gfCNCPoint1[8476] = {X 60.5656, Y 8.0531, Z -1.3333, A 0.000, B 0.000, C 0.000 }
gfCNCPoint1[8477] = {X 61.4618, Y 8.3667, Z -1.3333, A 0.000, B 0.000, C 0.000 }
gfCNCPoint1[8478] = {X 62.2657, Y 8.8718, Z -1.3333, A 0.000, B 0.000, C 0.000 }
gfCNCPoint1[8479] = {X 62.9371, Y 9.5432, Z -1.3333, A 0.000, B 0.000, C 0.000 }
gfCNCPoint1[8480] = {X 63.4422, Y 10.3471, Z -1.3333, A 0.000, B 0.000, C 0.000 }
gfCNCPoint1[8481] = {X 63.7558, Y 11.2433, Z -1.3333, A 0.000, B 0.000, C 0.000 }
gfCNCPoint1[8482] = {X 63.8621, Y 12.1868, Z -1.3333, A 0.000, B 0.000, C 0.000 }
gfCNCPoint1[8483] = {X 63.8621, Y 12.9781, Z -1.3333, A 0.000, B 0.000, C 0.000 }
gfCNCPoint1[8484] = {X 63.7771, Y 13.8227, Z -1.3333, A 0.000, B 0.000, C 0.000 }
gfCNCPoint1[8485] = {X 63.5256, Y 14.6335, Z -1.3333, A 0.000, B 0.000, C 0.000 }
gfCNCPoint1[8486] = {X 63.1176, Y 15.3779, Z -1.3333, A 0.000, B 0.000, C 0.000 }
gfCNCPoint1[8487] = {X 63.3949, Y 16.1022, Z -1.3333, A 0.000, B 0.000, C 0.000 }
gfCNCPoint1[8488] = {X 65.9589, Y 22.9155, Z -1.3333, A 0.000, B 0.000, C 0.000 }
gfCNCPoint1[8489] = {X 72.1337, Y 39.5291, Z -1.3333, A 0.000, B 0.000, C 0.000 }
gfCNCPoint1[8490] = {X 72.4511, Y 40.3274, Z -1.3333, A 0.000, B 0.000, C 0.000 }
gfCNCPoint1[8491] = {X 73.2892, Y 40.8174, Z -1.3333, A 0.000, B 0.000, C 0.000 }
gfCNCPoint1[8492] = {X 73.9939, Y 41.4851, Z -1.3333, A 0.000, B 0.000, C 0.000 }
gfCNCPoint1[8493] = {X 74.5283, Y 42.2956, Z -1.3333, A 0.000, B 0.000, C 0.000 }
gfCNCPoint1[8494] = {X 74.8643, Y 43.2065, Z -1.3333, A 0.000, B 0.000, C 0.000 }
gfCNCPoint1[8495] = {X 74.9843, Y 44.1699, Z -1.3333, A 0.000, B 0.000, C 0.000 }
gfCNCPoint1[8496] = {X 74.9845, Y 45.0000, Z -1.3333, A 0.000, B 0.000, C 0.000 }
gfCNCPoint1[8497] = {X 74.8782, Y 45.9435, Z -1.3333, A 0.000, B 0.000, C 0.000 }
gfCNCPoint1[8498] = {X 74.5646, Y 46.8397, Z -1.3333, A 0.000, B 0.000, C 0.000 }
gfCNCPoint1[8499] = {X 74.0594, Y 47.6436, Z -1.3333, A 0.000, B 0.000, C 0.000 }
gfCNCPoint1[8500] = {X 73.3881, Y 48.3150, Z -1.3333, A 0.000, B 0.000, C 0.000 }
gfCNCPoint1[8501] = {X 72.5841, Y 48.8201, Z -1.3333, A 0.000, B 0.000, C 0.000 }
gfCNCPoint1[8502] = {X 71.6879, Y 49.1337, Z -1.3333, A 0.000, B 0.000, C 0.000 }
gfCNCPoint1[8503] = {X 70.7445, Y 49.2400, Z -1.3333, A 0.000, B 0.000, C 0.000 }
gfCNCPoint1[8504] = {X 64.1851, Y 49.2400, Z -1.3333, A 0.000, B 0.000, C 0.000 }
gfCNCPoint1[8505] = {X 63.2416, Y 49.1337, Z -1.3333, A 0.000, B 0.000, C 0.000 }
gfCNCPoint1[8506] = {X 62.3455, Y 48.8201, Z -1.3333, A 0.000, B 0.000, C 0.000 }
gfCNCPoint1[8507] = {X 61.5415, Y 48.3150, Z -1.3333, A 0.000, B 0.000, C 0.000 }
gfCNCPoint1[8508] = {X 60.8702, Y 47.6436, Z -1.3333, A 0.000, B 0.000, C 0.000 }
gfCNCPoint1[8509] = {X 60.3650, Y 46.8397, Z -1.3333, A 0.000, B 0.000, C 0.000 }
gfCNCPoint1[8510] = {X 60.0514, Y 45.9435, Z -1.3333, A 0.000, B 0.000, C 0.000 }
gfCNCPoint1[8511] = {X 59.9451, Y 45.0000, Z -1.3333, A 0.000, B 0.000, C 0.000 }
gfCNCPoint1[8512] = {X 59.9451, Y 44.2085, Z -1.3333, A 0.000, B 0.000, C 0.000 }
gfCNCPoint1[8513] = {X 60.0333, Y 43.3524, Z -1.3333, A 0.000, B 0.000, C 0.000 }
gfCNCPoint1[8514] = {X 60.2925, Y 42.5318, Z -1.3333, A 0.000, B 0.000, C 0.000 }
gfCNCPoint1[8515] = {X 60.7121, Y 41.7805, Z -1.3333, A 0.000, B 0.000, C 0.000 }
gfCNCPoint1[8516] = {X 60.0634, Y 40.0092, Z -1.3333, A 0.000, B 0.000, C 0.000 }
gfCNCPoint1[8517] = {X 52.0206, Y 40.0092, Z -1.3333, A 0.000, B 0.000, C 0.000 }
gfCNCPoint1[8518] = {X 51.2452, Y 42.0920, Z -1.3333, A 0.000, B 0.000, C 0.000 }
gfCNCPoint1[8519] = {X 51.2680, Y 42.1293, Z -1.3333, A 0.000, B 0.000, C 0.000 }
gfCNCPoint1[8520] = {X 51.5637, Y 42.7765, Z -1.3333, A 0.000, B 0.000, C 0.000 }
gfCNCPoint1[8521] = {X 51.7470, Y 43.4641, Z -1.3333, A 0.000, B 0.000, C 0.000 }
gfCNCPoint1[8522] = {X 51.8128, Y 44.1726, Z -1.3333, A 0.000, B 0.000, C 0.000 }
gfCNCPoint1[8523] = {X 51.8129, Y 45.0000, Z -1.3333, A 0.000, B 0.000, C 0.000 }
gfCNCPoint1[8524] = {X 51.7066, Y 45.9435, Z -1.3333, A 0.000, B 0.000, C 0.000 }
gfCNCPoint1[8525] = {X 51.3930, Y 46.8397, Z -1.3333, A 0.000, B 0.000, C 0.000 }
gfCNCPoint1[8526] = {X 50.8879, Y 47.6436, Z -1.3333, A 0.000, B 0.000, C 0.000 }
gfCNCPoint1[8527] = {X 50.2165, Y 48.3150, Z -1.3333, A 0.000, B 0.000, C 0.000 }
gfCNCPoint1[8528] = {X 49.4126, Y 48.8201, Z -1.3333, A 0.000, B 0.000, C 0.000 }
gfCNCPoint1[8529] = {X 48.5164, Y 49.1337, Z -1.3333, A 0.000, B 0.000, C 0.000 }
gfCNCPoint1[8530] = {X 47.5729, Y 49.2400, Z -1.3333, A 0.000, B 0.000, C 0.000 }
gfCNCPoint1[8531] = {X 40.6393, Y 49.2400, Z -1.3333, A 0.000, B 0.000, C 0.000 }
gfCNCPoint1[8532] = {X 39.6958, Y 49.1337, Z -1.3333, A 0.000, B 0.000, C 0.000 }
gfCNCPoint1[8533] = {X 38.7996, Y 48.8201, Z -1.3333, A 0.000, B 0.000, C 0.000 }
gfCNCPoint1[8534] = {X 37.9957, Y 48.3150, Z -1.3333, A 0.000, B 0.000, C 0.000 }
gfCNCPoint1[8535] = {X 37.3243, Y 47.6436, Z -1.3333, A 0.000, B 0.000, C 0.000 }
gfCNCPoint1[8536] = {X 36.8192, Y 46.8397, Z -1.3333, A 0.000, B 0.000, C 0.000 }
gfCNCPoint1[8537] = {X 36.5056, Y 45.9435, Z -1.3333, A 0.000, B 0.000, C 0.000 }
gfCNCPoint1[8538] = {X 36.3993, Y 45.0000, Z -1.3333, A 0.000, B 0.000, C 0.000 }
gfCNCPoint1[8539] = {X 36.3993, Y 44.2086, Z -1.3333, A 0.000, B 0.000, C 0.000 }
gfCNCPoint1[8540] = {X 36.5154, Y 43.2237, Z -1.3333, A 0.000, B 0.000, C 0.000 }
gfCNCPoint1[8541] = {X 36.8572, Y 42.2926, Z -1.3333, A 0.000, B 0.000, C 0.000 }
gfCNCPoint1[8542] = {X 37.4059, Y 41.4664, Z -1.3333, A 0.000, B 0.000, C 0.000 }
gfCNCPoint1[8543] = {X 38.1315, Y 40.7903, Z -1.3333, A 0.000, B 0.000, C 0.000 }
gfCNCPoint1[8544] = {X 38.9944, Y 40.3012, Z -1.3333, A 0.000, B 0.000, C 0.000 }
gfCNCPoint1[8545] = {X 39.5929, Y 38.8890, Z -1.3333, A 0.000, B 0.000, C 0.000 }
gfCNCPoint1[8546] = {X 40.1409, Y 37.4565, Z -1.3333, A 0.000, B 0.000, C 0.000 }
gfCNCPoint1[8547] = {X 43.7241, Y 27.8349, Z -1.3333, A 0.000, B 0.000, C 0.000 }
gfCNCPoint1[8548] = {X 39.9756, Y 26.4389, Z -1.3333, A 0.000, B 0.000, C 0.000 }
gfCNCPoint1[8549] = {X 43.7991, Y 27.8628, Z -1.3333, A 0.000, B 0.000, C 0.000 }
gfCNCPoint1[8550] = {X 48.4687, Y 15.3238, Z -1.3333, A 0.000, B 0.000, C 0.000 }
gfCNCPoint1[8551] = {X 48.0765, Y 14.6072, Z -1.3333, A 0.000, B 0.000, C 0.000 }
gfCNCPoint1[8552] = {X 47.8320, Y 13.8278, Z -1.3333, A 0.000, B 0.000, C 0.000 }
gfCNCPoint1[8553] = {X 47.7444, Y 13.0157, Z -1.3333, A 0.000, B 0.000, C 0.000 }
gfCNCPoint1[8554] = {X 47.7442, Y 12.1868, Z -1.3333, A 0.000, B 0.000, C 0.000 }
gfCNCPoint1[8555] = {X 47.8485, Y 11.2611, Z -1.3333, A 0.000, B 0.000, C 0.000 }
gfCNCPoint1[8556] = {X 48.1562, Y 10.3819, Z -1.3333, A 0.000, B 0.000, C 0.000 }
gfCNCPoint1[8557] = {X 48.6518, Y 9.5931, Z -1.3333, A 0.000, B 0.000, C 0.000 }
gfCNCPoint1[8558] = {X 49.3105, Y 8.9344, Z -1.3333, A 0.000, B 0.000, C 0.000 }
gfCNCPoint1[8559] = {X 50.0993, Y 8.4388, Z -1.3333, A 0.000, B 0.000, C 0.000 }
gfCNCPoint1[8560] = {X 50.9785, Y 8.1311, Z -1.3333, A 0.000, B 0.000, C 0.000 }
gfCNCPoint1[8561] = {X 51.9042, Y 8.0268, Z -1.3333, A 0.000, B 0.000, C 0.000 }
gfCNCPoint1[8562] = {X 59.6221, Y 8.0268, Z -1.3333, A 0.000, B 0.000, C 0.000 }
gfCNCPoint1[8563] = {X 60.5478, Y 8.1311, Z -1.3333, A 0.000, B 0.000, C 0.000 }
gfCNCPoint1[8564] = {X 61.4271, Y 8.4388, Z -1.3333, A 0.000, B 0.000, C 0.000 }
gfCNCPoint1[8565] = {X 62.2158, Y 8.9344, Z -1.3333, A 0.000, B 0.000, C 0.000 }
gfCNCPoint1[8566] = {X 62.8745, Y 9.5931, Z -1.3333, A 0.000, B 0.000, C 0.000 }
gfCNCPoint1[8567] = {X 63.3702, Y 10.3819, Z -1.3333, A 0.000, B 0.000, C 0.000 }
gfCNCPoint1[8568] = {X 63.6778, Y 11.2611, Z -1.3333, A 0.000, B 0.000, C 0.000 }
gfCNCPoint1[8569] = {X 63.7821, Y 12.1868, Z -1.3333, A 0.000, B 0.000, C 0.000 }
gfCNCPoint1[8570] = {X 63.7821, Y 12.9781, Z -1.3333, A 0.000, B 0.000, C 0.000 }
gfCNCPoint1[8571] = {X 63.6959, Y 13.8205, Z -1.3333, A 0.000, B 0.000, C 0.000 }
gfCNCPoint1[8572] = {X 63.4410, Y 14.6279, Z -1.3333, A 0.000, B 0.000, C 0.000 }
gfCNCPoint1[8573] = {X 63.0278, Y 15.3670, Z -1.3333, A 0.000, B 0.000, C 0.000 }
gfCNCPoint1[8574] = {X 63.3201, Y 16.1306, Z -1.3333, A 0.000, B 0.000, C 0.000 }
gfCNCPoint1[8575] = {X 65.8840, Y 22.9436, Z -1.3333, A 0.000, B 0.000, C 0.000 }
gfCNCPoint1[8576] = {X 72.0590, Y 39.5578, Z -1.3333, A 0.000, B 0.000, C 0.000 }
gfCNCPoint1[8577] = {X 72.3889, Y 40.3876, Z -1.3333, A 0.000, B 0.000, C 0.000 }
gfCNCPoint1[8578] = {X 73.2202, Y 40.8657, Z -1.3333, A 0.000, B 0.000, C 0.000 }
gfCNCPoint1[8579] = {X 73.9200, Y 41.5215, Z -1.3333, A 0.000, B 0.000, C 0.000 }
gfCNCPoint1[8580] = {X 74.4510, Y 42.3201, Z -1.3333, A 0.000, B 0.000, C 0.000 }
gfCNCPoint1[8581] = {X 74.7850, Y 43.2191, Z -1.3333, A 0.000, B 0.000, C 0.000 }
gfCNCPoint1[8582] = {X 74.9043, Y 44.1706, Z -1.3333, A 0.000, B 0.000, C 0.000 }
gfCNCPoint1[8583] = {X 74.9045, Y 45.0000, Z -1.3333, A 0.000, B 0.000, C 0.000 }
gfCNCPoint1[8584] = {X 74.8002, Y 45.9257, Z -1.3333, A 0.000, B 0.000, C 0.000 }
gfCNCPoint1[8585] = {X 74.4925, Y 46.8050, Z -1.3333, A 0.000, B 0.000, C 0.000 }
gfCNCPoint1[8586] = {X 73.9969, Y 47.5937, Z -1.3333, A 0.000, B 0.000, C 0.000 }
gfCNCPoint1[8587] = {X 73.3382, Y 48.2524, Z -1.3333, A 0.000, B 0.000, C 0.000 }
gfCNCPoint1[8588] = {X 72.5494, Y 48.7480, Z -1.3333, A 0.000, B 0.000, C 0.000 }
gfCNCPoint1[8589] = {X 71.6701, Y 49.0557, Z -1.3333, A 0.000, B 0.000, C 0.000 }
gfCNCPoint1[8590] = {X 70.7445, Y 49.1600, Z -1.3333, A 0.000, B 0.000, C 0.000 }
gfCNCPoint1[8591] = {X 64.1851, Y 49.1600, Z -1.3333, A 0.000, B 0.000, C 0.000 }
gfCNCPoint1[8592] = {X 63.2594, Y 49.0557, Z -1.3333, A 0.000, B 0.000, C 0.000 }
gfCNCPoint1[8593] = {X 62.3802, Y 48.7480, Z -1.3333, A 0.000, B 0.000, C 0.000 }
gfCNCPoint1[8594] = {X 61.5914, Y 48.2524, Z -1.3333, A 0.000, B 0.000, C 0.000 }
gfCNCPoint1[8595] = {X 60.9327, Y 47.5937, Z -1.3333, A 0.000, B 0.000, C 0.000 }
gfCNCPoint1[8596] = {X 60.4371, Y 46.8050, Z -1.3333, A 0.000, B 0.000, C 0.000 }
gfCNCPoint1[8597] = {X 60.1294, Y 45.9257, Z -1.3333, A 0.000, B 0.000, C 0.000 }
gfCNCPoint1[8598] = {X 60.0251, Y 45.0000, Z -1.3333, A 0.000, B 0.000, C 0.000 }
gfCNCPoint1[8599] = {X 60.0251, Y 44.2086, Z -1.3333, A 0.000, B 0.000, C 0.000 }
gfCNCPoint1[8600] = {X 60.1145, Y 43.3551, Z -1.3333, A 0.000, B 0.000, C 0.000 }
gfCNCPoint1[8601] = {X 60.3770, Y 42.5381, Z -1.3333, A 0.000, B 0.000, C 0.000 }
gfCNCPoint1[8602] = {X 60.8017, Y 41.7924, Z -1.3333, A 0.000, B 0.000, C 0.000 }
gfCNCPoint1[8603] = {X 60.1193, Y 39.9292, Z -1.3333, A 0.000, B 0.000, C 0.000 }
gfCNCPoint1[8604] = {X 51.9650, Y 39.9292, Z -1.3333, A 0.000, B 0.000, C 0.000 }
gfCNCPoint1[8605] = {X 51.1567, Y 42.1005, Z -1.3333, A 0.000, B 0.000, C 0.000 }
gfCNCPoint1[8606] = {X 51.1989, Y 42.1698, Z -1.3333, A 0.000, B 0.000, C 0.000 }
gfCNCPoint1[8607] = {X 51.4887, Y 42.8044, Z -1.3333, A 0.000, B 0.000, C 0.000 }
gfCNCPoint1[8608] = {X 51.6683, Y 43.4786, Z -1.3333, A 0.000, B 0.000, C 0.000 }
gfCNCPoint1[8609] = {X 51.7328, Y 44.1733, Z -1.3333, A 0.000, B 0.000, C 0.000 }
gfCNCPoint1[8610] = {X 51.7329, Y 45.0000, Z -1.3333, A 0.000, B 0.000, C 0.000 }
gfCNCPoint1[8611] = {X 51.6286, Y 45.9257, Z -1.3333, A 0.000, B 0.000, C 0.000 }
gfCNCPoint1[8612] = {X 51.3210, Y 46.8050, Z -1.3333, A 0.000, B 0.000, C 0.000 }
gfCNCPoint1[8613] = {X 50.8253, Y 47.5937, Z -1.3333, A 0.000, B 0.000, C 0.000 }
gfCNCPoint1[8614] = {X 50.1666, Y 48.2524, Z -1.3333, A 0.000, B 0.000, C 0.000 }
gfCNCPoint1[8615] = {X 49.3779, Y 48.7480, Z -1.3333, A 0.000, B 0.000, C 0.000 }
gfCNCPoint1[8616] = {X 48.4986, Y 49.0557, Z -1.3333, A 0.000, B 0.000, C 0.000 }
gfCNCPoint1[8617] = {X 47.5729, Y 49.1600, Z -1.3333, A 0.000, B 0.000, C 0.000 }
gfCNCPoint1[8618] = {X 40.6393, Y 49.1600, Z -1.3333, A 0.000, B 0.000, C 0.000 }
gfCNCPoint1[8619] = {X 39.7136, Y 49.0557, Z -1.3333, A 0.000, B 0.000, C 0.000 }
gfCNCPoint1[8620] = {X 38.8343, Y 48.7480, Z -1.3333, A 0.000, B 0.000, C 0.000 }
gfCNCPoint1[8621] = {X 38.0456, Y 48.2524, Z -1.3333, A 0.000, B 0.000, C 0.000 }
gfCNCPoint1[8622] = {X 37.3869, Y 47.5937, Z -1.3333, A 0.000, B 0.000, C 0.000 }
gfCNCPoint1[8623] = {X 36.8913, Y 46.8050, Z -1.3333, A 0.000, B 0.000, C 0.000 }
gfCNCPoint1[8624] = {X 36.5836, Y 45.9257, Z -1.3333, A 0.000, B 0.000, C 0.000 }
gfCNCPoint1[8625] = {X 36.4793, Y 45.0000, Z -1.3333, A 0.000, B 0.000, C 0.000 }
gfCNCPoint1[8626] = {X 36.4793, Y 44.2087, Z -1.3333, A 0.000, B 0.000, C 0.000 }
gfCNCPoint1[8627] = {X 36.5947, Y 43.2361, Z -1.3333, A 0.000, B 0.000, C 0.000 }
gfCNCPoint1[8628] = {X 36.9343, Y 42.3175, Z -1.3333, A 0.000, B 0.000, C 0.000 }
gfCNCPoint1[8629] = {X 37.4792, Y 41.5038, Z -1.3333, A 0.000, B 0.000, C 0.000 }
gfCNCPoint1[8630] = {X 38.1992, Y 40.8399, Z -1.3333, A 0.000, B 0.000, C 0.000 }
gfCNCPoint1[8631] = {X 39.0545, Y 40.3629, Z -1.3333, A 0.000, B 0.000, C 0.000 }
gfCNCPoint1[8632] = {X 39.6611, Y 38.9337, Z -1.3333, A 0.000, B 0.000, C 0.000 }
gfCNCPoint1[8633] = {X 40.2162, Y 37.4838, Z -1.3333, A 0.000, B 0.000, C 0.000 }
gfCNCPoint1[8634] = {X 43.7991, Y 27.8628, Z -1.3333, A 0.000, B 0.000, C 0.000 }
gfCNCPoint1[8635] = {X 40.0506, Y 26.4668, Z -1.3333, A 0.000, B 0.000, C 0.000 }
gfCNCPoint1[8636] = {X 43.8740, Y 27.8907, Z -1.3333, A 0.000, B 0.000, C 0.000 }
gfCNCPoint1[8637] = {X 48.5582, Y 15.3126, Z -1.3333, A 0.000, B 0.000, C 0.000 }
gfCNCPoint1[8638] = {X 48.1610, Y 14.6012, Z -1.3333, A 0.000, B 0.000, C 0.000 }
gfCNCPoint1[8639] = {X 47.9131, Y 13.8250, Z -1.3333, A 0.000, B 0.000, C 0.000 }
gfCNCPoint1[8640] = {X 47.8244, Y 13.0150, Z -1.3333, A 0.000, B 0.000, C 0.000 }
gfCNCPoint1[8641] = {X 47.8242, Y 12.1868, Z -1.3333, A 0.000, B 0.000, C 0.000 }
gfCNCPoint1[8642] = {X 47.9265, Y 11.2789, Z -1.3333, A 0.000, B 0.000, C 0.000 }
gfCNCPoint1[8643] = {X 48.2283, Y 10.4166, Z -1.3333, A 0.000, B 0.000, C 0.000 }
gfCNCPoint1[8644] = {X 48.7144, Y 9.6430, Z -1.3333, A 0.000, B 0.000, C 0.000 }
gfCNCPoint1[8645] = {X 49.3604, Y 8.9969, Z -1.3333, A 0.000, B 0.000, C 0.000 }
gfCNCPoint1[8646] = {X 50.1340, Y 8.5109, Z -1.3333, A 0.000, B 0.000, C 0.000 }
gfCNCPoint1[8647] = {X 50.9963, Y 8.2091, Z -1.3333, A 0.000, B 0.000, C 0.000 }
gfCNCPoint1[8648] = {X 51.9042, Y 8.1068, Z -1.3333, A 0.000, B 0.000, C 0.000 }
gfCNCPoint1[8649] = {X 59.6221, Y 8.1068, Z -1.3333, A 0.000, B 0.000, C 0.000 }
gfCNCPoint1[8650] = {X 60.5300, Y 8.2091, Z -1.3333, A 0.000, B 0.000, C 0.000 }
gfCNCPoint1[8651] = {X 61.3924, Y 8.5109, Z -1.3333, A 0.000, B 0.000, C 0.000 }
gfCNCPoint1[8652] = {X 62.1660, Y 8.9969, Z -1.3333, A 0.000, B 0.000, C 0.000 }
gfCNCPoint1[8653] = {X 62.8120, Y 9.6430, Z -1.3333, A 0.000, B 0.000, C 0.000 }
gfCNCPoint1[8654] = {X 63.2981, Y 10.4166, Z -1.3333, A 0.000, B 0.000, C 0.000 }
gfCNCPoint1[8655] = {X 63.5998, Y 11.2789, Z -1.3333, A 0.000, B 0.000, C 0.000 }
gfCNCPoint1[8656] = {X 63.7021, Y 12.1868, Z -1.3333, A 0.000, B 0.000, C 0.000 }
gfCNCPoint1[8657] = {X 63.7021, Y 12.9781, Z -1.3333, A 0.000, B 0.000, C 0.000 }
gfCNCPoint1[8658] = {X 63.6147, Y 13.8181, Z -1.3333, A 0.000, B 0.000, C 0.000 }
gfCNCPoint1[8659] = {X 63.3562, Y 14.6221, Z -1.3333, A 0.000, B 0.000, C 0.000 }
gfCNCPoint1[8660] = {X 62.9377, Y 15.3556, Z -1.3333, A 0.000, B 0.000, C 0.000 }
gfCNCPoint1[8661] = {X 63.2453, Y 16.1590, Z -1.3333, A 0.000, B 0.000, C 0.000 }
gfCNCPoint1[8662] = {X 65.8090, Y 22.9716, Z -1.3333, A 0.000, B 0.000, C 0.000 }
gfCNCPoint1[8663] = {X 71.9843, Y 39.5865, Z -1.3333, A 0.000, B 0.000, C 0.000 }
gfCNCPoint1[8664] = {X 72.3269, Y 40.4482, Z -1.3333, A 0.000, B 0.000, C 0.000 }
gfCNCPoint1[8665] = {X 73.1513, Y 40.9144, Z -1.3333, A 0.000, B 0.000, C 0.000 }
gfCNCPoint1[8666] = {X 73.8461, Y 41.5581, Z -1.3333, A 0.000, B 0.000, C 0.000 }
gfCNCPoint1[8667] = {X 74.3737, Y 42.3446, Z -1.3333, A 0.000, B 0.000, C 0.000 }
gfCNCPoint1[8668] = {X 74.7057, Y 43.2317, Z -1.3333, A 0.000, B 0.000, C 0.000 }
gfCNCPoint1[8669] = {X 74.8243, Y 44.1714, Z -1.3333, A 0.000, B 0.000, C 0.000 }
gfCNCPoint1[8670] = {X 74.8245, Y 45.0000, Z -1.3333, A 0.000, B 0.000, C 0.000 }
gfCNCPoint1[8671] = {X 74.7222, Y 45.9079, Z -1.3333, A 0.000, B 0.000, C 0.000 }
gfCNCPoint1[8672] = {X 74.4204, Y 46.7702, Z -1.3333, A 0.000, B 0.000, C 0.000 }
gfCNCPoint1[8673] = {X 73.9343, Y 47.5438, Z -1.3333, A 0.000, B 0.000, C 0.000 }
gfCNCPoint1[8674] = {X 73.2883, Y 48.1899, Z -1.3333, A 0.000, B 0.000, C 0.000 }
gfCNCPoint1[8675] = {X 72.5147, Y 48.6760, Z -1.3333, A 0.000, B 0.000, C 0.000 }
gfCNCPoint1[8676] = {X 71.6523, Y 48.9777, Z -1.3333, A 0.000, B 0.000, C 0.000 }
gfCNCPoint1[8677] = {X 70.7445, Y 49.0800, Z -1.3333, A 0.000, B 0.000, C 0.000 }
gfCNCPoint1[8678] = {X 64.1851, Y 49.0800, Z -1.3333, A 0.000, B 0.000, C 0.000 }
gfCNCPoint1[8679] = {X 63.2772, Y 48.9777, Z -1.3333, A 0.000, B 0.000, C 0.000 }
gfCNCPoint1[8680] = {X 62.4149, Y 48.6760, Z -1.3333, A 0.000, B 0.000, C 0.000 }
gfCNCPoint1[8681] = {X 61.6413, Y 48.1899, Z -1.3333, A 0.000, B 0.000, C 0.000 }
gfCNCPoint1[8682] = {X 60.9953, Y 47.5438, Z -1.3333, A 0.000, B 0.000, C 0.000 }
gfCNCPoint1[8683] = {X 60.5092, Y 46.7702, Z -1.3333, A 0.000, B 0.000, C 0.000 }
gfCNCPoint1[8684] = {X 60.2074, Y 45.9079, Z -1.3333, A 0.000, B 0.000, C 0.000 }
gfCNCPoint1[8685] = {X 60.1051, Y 45.0000, Z -1.3333, A 0.000, B 0.000, C 0.000 }
gfCNCPoint1[8686] = {X 60.1051, Y 44.2087, Z -1.3333, A 0.000, B 0.000, C 0.000 }
gfCNCPoint1[8687] = {X 60.1957, Y 43.3579, Z -1.3333, A 0.000, B 0.000, C 0.000 }
gfCNCPoint1[8688] = {X 60.4617, Y 42.5447, Z -1.3333, A 0.000, B 0.000, C 0.000 }
gfCNCPoint1[8689] = {X 60.8914, Y 41.8048, Z -1.3333, A 0.000, B 0.000, C 0.000 }
gfCNCPoint1[8690] = {X 60.1752, Y 39.8492, Z -1.3333, A 0.000, B 0.000, C 0.000 }
gfCNCPoint1[8691] = {X 51.9094, Y 39.8492, Z -1.3333, A 0.000, B 0.000, C 0.000 }
gfCNCPoint1[8692] = {X 51.0681, Y 42.1090, Z -1.3333, A 0.000, B 0.000, C 0.000 }
gfCNCPoint1[8693] = {X 51.1306, Y 42.2115, Z -1.3333, A 0.000, B 0.000, C 0.000 }
gfCNCPoint1[8694] = {X 51.4141, Y 42.8332, Z -1.3333, A 0.000, B 0.000, C 0.000 }
gfCNCPoint1[8695] = {X 51.5898, Y 43.4936, Z -1.3333, A 0.000, B 0.000, C 0.000 }
gfCNCPoint1[8696] = {X 51.6528, Y 44.1740, Z -1.3333, A 0.000, B 0.000, C 0.000 }
gfCNCPoint1[8697] = {X 51.6529, Y 45.0000, Z -1.3333, A 0.000, B 0.000, C 0.000 }
gfCNCPoint1[8698] = {X 51.5506, Y 45.9079, Z -1.3333, A 0.000, B 0.000, C 0.000 }
gfCNCPoint1[8699] = {X 51.2489, Y 46.7702, Z -1.3333, A 0.000, B 0.000, C 0.000 }
gfCNCPoint1[8700] = {X 50.7628, Y 47.5438, Z -1.3333, A 0.000, B 0.000, C 0.000 }
gfCNCPoint1[8701] = {X 50.1168, Y 48.1899, Z -1.3333, A 0.000, B 0.000, C 0.000 }
gfCNCPoint1[8702] = {X 49.3432, Y 48.6760, Z -1.3333, A 0.000, B 0.000, C 0.000 }
gfCNCPoint1[8703] = {X 48.4808, Y 48.9777, Z -1.3333, A 0.000, B 0.000, C 0.000 }
gfCNCPoint1[8704] = {X 47.5729, Y 49.0800, Z -1.3333, A 0.000, B 0.000, C 0.000 }
gfCNCPoint1[8705] = {X 40.6393, Y 49.0800, Z -1.3333, A 0.000, B 0.000, C 0.000 }
gfCNCPoint1[8706] = {X 39.7314, Y 48.9777, Z -1.3333, A 0.000, B 0.000, C 0.000 }
gfCNCPoint1[8707] = {X 38.8691, Y 48.6760, Z -1.3333, A 0.000, B 0.000, C 0.000 }
gfCNCPoint1[8708] = {X 38.0955, Y 48.1899, Z -1.3333, A 0.000, B 0.000, C 0.000 }
gfCNCPoint1[8709] = {X 37.4494, Y 47.5438, Z -1.3333, A 0.000, B 0.000, C 0.000 }
gfCNCPoint1[8710] = {X 36.9633, Y 46.7702, Z -1.3333, A 0.000, B 0.000, C 0.000 }
gfCNCPoint1[8711] = {X 36.6616, Y 45.9079, Z -1.3333, A 0.000, B 0.000, C 0.000 }
gfCNCPoint1[8712] = {X 36.5593, Y 45.0000, Z -1.3333, A 0.000, B 0.000, C 0.000 }
gfCNCPoint1[8713] = {X 36.5593, Y 44.2087, Z -1.3333, A 0.000, B 0.000, C 0.000 }
gfCNCPoint1[8714] = {X 36.6682, Y 43.2722, Z -1.3333, A 0.000, B 0.000, C 0.000 }
gfCNCPoint1[8715] = {X 36.9892, Y 42.3858, Z -1.3333, A 0.000, B 0.000, C 0.000 }
gfCNCPoint1[8716] = {X 37.5050, Y 41.5968, Z -1.3333, A 0.000, B 0.000, C 0.000 }
gfCNCPoint1[8717] = {X 38.1882, Y 40.9471, Z -1.3333, A 0.000, B 0.000, C 0.000 }
gfCNCPoint1[8718] = {X 39.0022, Y 40.4716, Z -1.3333, A 0.000, B 0.000, C 0.000 }
gfCNCPoint1[8719] = {X 39.1147, Y 40.4243, Z -1.3333, A 0.000, B 0.000, C 0.000 }
gfCNCPoint1[8720] = {X 39.7294, Y 38.9783, Z -1.3333, A 0.000, B 0.000, C 0.000 }
gfCNCPoint1[8721] = {X 40.2914, Y 37.5110, Z -1.3333, A 0.000, B 0.000, C 0.000 }
gfCNCPoint1[8722] = {X 43.8740, Y 27.8907, Z -1.3333, A 0.000, B 0.000, C 0.000 }
gfCNCPoint1[8723] = {X 40.1255, Y 26.4948, Z -1.3333, A 0.000, B 0.000, C 0.000 }
gfCNCPoint1[8724] = {X 43.9490, Y 27.9186, Z -1.3333, A 0.000, B 0.000, C 0.000 }
gfCNCPoint1[8725] = {X 48.6479, Y 15.3010, Z -1.3333, A 0.000, B 0.000, C 0.000 }
gfCNCPoint1[8726] = {X 48.2407, Y 14.5838, Z -1.3333, A 0.000, B 0.000, C 0.000 }
gfCNCPoint1[8727] = {X 47.9892, Y 13.7983, Z -1.3333, A 0.000, B 0.000, C 0.000 }
gfCNCPoint1[8728] = {X 47.9042, Y 12.9779, Z -1.3333, A 0.000, B 0.000, C 0.000 }
gfCNCPoint1[8729] = {X 47.9042, Y 12.1868, Z -1.3333, A 0.000, B 0.000, C 0.000 }
gfCNCPoint1[8730] = {X 48.0045, Y 11.2967, Z -1.3333, A 0.000, B 0.000, C 0.000 }
gfCNCPoint1[8731] = {X 48.3003, Y 10.4513, Z -1.3333, A 0.000, B 0.000, C 0.000 }
gfCNCPoint1[8732] = {X 48.7769, Y 9.6929, Z -1.3333, A 0.000, B 0.000, C 0.000 }
gfCNCPoint1[8733] = {X 49.4103, Y 9.0595, Z -1.3333, A 0.000, B 0.000, C 0.000 }
gfCNCPoint1[8734] = {X 50.1687, Y 8.5829, Z -1.3333, A 0.000, B 0.000, C 0.000 }
gfCNCPoint1[8735] = {X 51.0141, Y 8.2871, Z -1.3333, A 0.000, B 0.000, C 0.000 }
gfCNCPoint1[8736] = {X 51.9042, Y 8.1868, Z -1.3333, A 0.000, B 0.000, C 0.000 }
gfCNCPoint1[8737] = {X 59.6221, Y 8.1868, Z -1.3333, A 0.000, B 0.000, C 0.000 }
gfCNCPoint1[8738] = {X 60.5122, Y 8.2871, Z -1.3333, A 0.000, B 0.000, C 0.000 }
gfCNCPoint1[8739] = {X 61.3577, Y 8.5829, Z -1.3333, A 0.000, B 0.000, C 0.000 }
gfCNCPoint1[8740] = {X 62.1161, Y 9.0595, Z -1.3333, A 0.000, B 0.000, C 0.000 }
gfCNCPoint1[8741] = {X 62.7495, Y 9.6929, Z -1.3333, A 0.000, B 0.000, C 0.000 }
gfCNCPoint1[8742] = {X 63.2260, Y 10.4513, Z -1.3333, A 0.000, B 0.000, C 0.000 }
gfCNCPoint1[8743] = {X 63.5218, Y 11.2967, Z -1.3333, A 0.000, B 0.000, C 0.000 }
gfCNCPoint1[8744] = {X 63.6221, Y 12.1868, Z -1.3333, A 0.000, B 0.000, C 0.000 }
gfCNCPoint1[8745] = {X 63.6219, Y 13.0192, Z -1.3333, A 0.000, B 0.000, C 0.000 }
gfCNCPoint1[8746] = {X 63.5276, Y 13.8424, Z -1.3333, A 0.000, B 0.000, C 0.000 }
gfCNCPoint1[8747] = {X 63.2657, Y 14.6285, Z -1.3333, A 0.000, B 0.000, C 0.000 }
gfCNCPoint1[8748] = {X 62.8475, Y 15.3438, Z -1.3333, A 0.000, B 0.000, C 0.000 }
gfCNCPoint1[8749] = {X 63.1705, Y 16.1874, Z -1.3333, A 0.000, B 0.000, C 0.000 }
gfCNCPoint1[8750] = {X 65.7341, Y 22.9996, Z -1.3333, A 0.000, B 0.000, C 0.000 }
gfCNCPoint1[8751] = {X 71.9097, Y 39.6152, Z -1.3333, A 0.000, B 0.000, C 0.000 }
gfCNCPoint1[8752] = {X 72.2605, Y 40.4978, Z -1.3333, A 0.000, B 0.000, C 0.000 }
gfCNCPoint1[8753] = {X 72.2762, Y 40.5137, Z -1.3333, A 0.000, B 0.000, C 0.000 }
gfCNCPoint1[8754] = {X 72.3430, Y 40.5421, Z -1.3333, A 0.000, B 0.000, C 0.000 }
gfCNCPoint1[8755] = {X 72.4093, Y 40.5717, Z -1.3333, A 0.000, B 0.000, C 0.000 }
gfCNCPoint1[8756] = {X 73.1893, Y 41.0429, Z -1.3333, A 0.000, B 0.000, C 0.000 }
gfCNCPoint1[8757] = {X 73.8424, Y 41.6784, Z -1.3333, A 0.000, B 0.000, C 0.000 }
gfCNCPoint1[8758] = {X 74.3347, Y 42.4452, Z -1.3333, A 0.000, B 0.000, C 0.000 }
gfCNCPoint1[8759] = {X 74.6407, Y 43.3036, Z -1.3333, A 0.000, B 0.000, C 0.000 }
gfCNCPoint1[8760] = {X 74.7445, Y 44.2089, Z -1.3333, A 0.000, B 0.000, C 0.000 }
gfCNCPoint1[8761] = {X 74.7445, Y 45.0000, Z -1.3333, A 0.000, B 0.000, C 0.000 }
gfCNCPoint1[8762] = {X 74.6442, Y 45.8901, Z -1.3333, A 0.000, B 0.000, C 0.000 }
gfCNCPoint1[8763] = {X 74.3483, Y 46.7355, Z -1.3333, A 0.000, B 0.000, C 0.000 }
gfCNCPoint1[8764] = {X 73.8718, Y 47.4940, Z -1.3333, A 0.000, B 0.000, C 0.000 }
gfCNCPoint1[8765] = {X 73.2384, Y 48.1273, Z -1.3333, A 0.000, B 0.000, C 0.000 }
gfCNCPoint1[8766] = {X 72.4800, Y 48.6039, Z -1.3333, A 0.000, B 0.000, C 0.000 }
gfCNCPoint1[8767] = {X 71.6345, Y 48.8997, Z -1.3333, A 0.000, B 0.000, C 0.000 }
gfCNCPoint1[8768] = {X 70.7445, Y 49.0000, Z -1.3333, A 0.000, B 0.000, C 0.000 }
gfCNCPoint1[8769] = {X 64.1851, Y 49.0000, Z -1.3333, A 0.000, B 0.000, C 0.000 }
gfCNCPoint1[8770] = {X 63.2951, Y 48.8997, Z -1.3333, A 0.000, B 0.000, C 0.000 }
gfCNCPoint1[8771] = {X 62.4496, Y 48.6039, Z -1.3333, A 0.000, B 0.000, C 0.000 }
gfCNCPoint1[8772] = {X 61.6912, Y 48.1273, Z -1.3333, A 0.000, B 0.000, C 0.000 }
gfCNCPoint1[8773] = {X 61.0578, Y 47.4940, Z -1.3333, A 0.000, B 0.000, C 0.000 }
gfCNCPoint1[8774] = {X 60.5813, Y 46.7355, Z -1.3333, A 0.000, B 0.000, C 0.000 }
gfCNCPoint1[8775] = {X 60.2854, Y 45.8901, Z -1.3333, A 0.000, B 0.000, C 0.000 }
gfCNCPoint1[8776] = {X 60.1851, Y 45.0000, Z -1.3333, A 0.000, B 0.000, C 0.000 }
gfCNCPoint1[8777] = {X 60.1855, Y 44.1538, Z -1.3333, A 0.000, B 0.000, C 0.000 }
gfCNCPoint1[8778] = {X 60.2746, Y 43.3674, Z -1.3333, A 0.000, B 0.000, C 0.000 }
gfCNCPoint1[8779] = {X 60.5168, Y 42.6140, Z -1.3333, A 0.000, B 0.000, C 0.000 }
gfCNCPoint1[8780] = {X 60.9025, Y 41.9231, Z -1.3333, A 0.000, B 0.000, C 0.000 }
gfCNCPoint1[8781] = {X 60.9815, Y 41.8181, Z -1.3333, A 0.000, B 0.000, C 0.000 }
gfCNCPoint1[8782] = {X 60.2311, Y 39.7692, Z -1.3333, A 0.000, B 0.000, C 0.000 }
gfCNCPoint1[8783] = {X 51.8417, Y 39.7692, Z -1.3333, A 0.000, B 0.000, C 0.000 }
gfCNCPoint1[8784] = {X 51.8417, Y 39.8018, Z -1.3333, A 0.000, B 0.000, C 0.000 }
gfCNCPoint1[8785] = {X 50.9796, Y 42.1175, Z -1.3333, A 0.000, B 0.000, C 0.000 }
gfCNCPoint1[8786] = {X 51.0718, Y 42.2703, Z -1.3333, A 0.000, B 0.000, C 0.000 }
gfCNCPoint1[8787] = {X 51.3476, Y 42.8851, Z -1.3333, A 0.000, B 0.000, C 0.000 }
gfCNCPoint1[8788] = {X 51.5162, Y 43.5375, Z -1.3333, A 0.000, B 0.000, C 0.000 }
gfCNCPoint1[8789] = {X 51.5729, Y 44.2089, Z -1.3333, A 0.000, B 0.000, C 0.000 }
gfCNCPoint1[8790] = {X 51.5729, Y 45.0000, Z -1.3333, A 0.000, B 0.000, C 0.000 }
gfCNCPoint1[8791] = {X 51.4726, Y 45.8901, Z -1.3333, A 0.000, B 0.000, C 0.000 }
gfCNCPoint1[8792] = {X 51.1768, Y 46.7355, Z -1.3333, A 0.000, B 0.000, C 0.000 }
gfCNCPoint1[8793] = {X 50.7003, Y 47.4940, Z -1.3333, A 0.000, B 0.000, C 0.000 }
gfCNCPoint1[8794] = {X 50.0669, Y 48.1273, Z -1.3333, A 0.000, B 0.000, C 0.000 }
gfCNCPoint1[8795] = {X 49.3085, Y 48.6039, Z -1.3333, A 0.000, B 0.000, C 0.000 }
gfCNCPoint1[8796] = {X 48.4630, Y 48.8997, Z -1.3333, A 0.000, B 0.000, C 0.000 }
gfCNCPoint1[8797] = {X 47.5729, Y 49.0000, Z -1.3333, A 0.000, B 0.000, C 0.000 }
gfCNCPoint1[8798] = {X 40.6393, Y 49.0000, Z -1.3333, A 0.000, B 0.000, C 0.000 }
gfCNCPoint1[8799] = {X 39.7492, Y 48.8997, Z -1.3333, A 0.000, B 0.000, C 0.000 }
gfCNCPoint1[8800] = {X 38.9038, Y 48.6039, Z -1.3333, A 0.000, B 0.000, C 0.000 }
gfCNCPoint1[8801] = {X 38.1453, Y 48.1273, Z -1.3333, A 0.000, B 0.000, C 0.000 }
gfCNCPoint1[8802] = {X 37.5120, Y 47.4940, Z -1.3333, A 0.000, B 0.000, C 0.000 }
gfCNCPoint1[8803] = {X 37.0354, Y 46.7355, Z -1.3333, A 0.000, B 0.000, C 0.000 }
gfCNCPoint1[8804] = {X 36.7396, Y 45.8901, Z -1.3333, A 0.000, B 0.000, C 0.000 }
gfCNCPoint1[8805] = {X 36.6393, Y 45.0000, Z -1.3333, A 0.000, B 0.000, C 0.000 }
gfCNCPoint1[8806] = {X 36.6397, Y 44.1538, Z -1.3333, A 0.000, B 0.000, C 0.000 }
gfCNCPoint1[8807] = {X 36.7564, Y 43.2479, Z -1.3333, A 0.000, B 0.000, C 0.000 }
gfCNCPoint1[8808] = {X 37.0756, Y 42.3922, Z -1.3333, A 0.000, B 0.000, C 0.000 }
gfCNCPoint1[8809] = {X 37.5806, Y 41.6311, Z -1.3333, A 0.000, B 0.000, C 0.000 }
gfCNCPoint1[8810] = {X 38.2450, Y 41.0045, Z -1.3333, A 0.000, B 0.000, C 0.000 }
gfCNCPoint1[8811] = {X 39.0343, Y 40.5449, Z -1.3333, A 0.000, B 0.000, C 0.000 }
gfCNCPoint1[8812] = {X 39.0895, Y 40.5212, Z -1.3333, A 0.000, B 0.000, C 0.000 }
gfCNCPoint1[8813] = {X 39.1451, Y 40.4984, Z -1.3333, A 0.000, B 0.000, C 0.000 }
gfCNCPoint1[8814] = {X 39.1703, Y 40.4820, Z -1.3333, A 0.000, B 0.000, C 0.000 }
gfCNCPoint1[8815] = {X 39.1875, Y 40.4575, Z -1.3333, A 0.000, B 0.000, C 0.000 }
gfCNCPoint1[8816] = {X 39.2136, Y 40.3990, Z -1.3333, A 0.000, B 0.000, C 0.000 }
gfCNCPoint1[8817] = {X 39.2395, Y 40.3406, Z -1.3333, A 0.000, B 0.000, C 0.000 }
gfCNCPoint1[8818] = {X 39.8274, Y 38.9492, Z -1.3333, A 0.000, B 0.000, C 0.000 }
gfCNCPoint1[8819] = {X 40.3666, Y 37.5383, Z -1.3333, A 0.000, B 0.000, C 0.000 }
gfCNCPoint1[8820] = {X 43.9490, Y 27.9186, Z -1.3333, A 0.000, B 0.000, C 0.000 }
gfCNCPoint1[8821] = {X 40.1255, Y 26.4948, Z -1.3333, A 0.000, B 0.000, C 0.000 }
gfCNCPoint1[8822] = {X 40.1255, Y 26.4948, Z 1.6667, A 0.000, B 0.000, C 0.000 }
gfCNCPoint1[8823] = {X 40.1255, Y 26.4948, Z 11.0000, A 0.000, B 0.000, C 0.000 }
gfCNCPoint1[8824] = {X 79.0239, Y 28.5924, Z 11.0000, A 0.000, B 0.000, C 0.000 }
gfCNCPoint1[8825] = {X 79.0239, Y 28.5924, Z 1.6667, A 0.000, B 0.000, C 0.000 }
gfCNCPoint1[8826] = {X 79.0239, Y 28.5924, Z -1.3333, A 0.000, B 0.000, C 0.000 }
gfCNCPoint1[8827] = {X 83.1039, Y 28.5924, Z -1.3333, A 0.000, B 0.000, C 0.000 }
gfCNCPoint1[8828] = {X 83.1037, Y 16.2751, Z -1.3333, A 0.000, B 0.000, C 0.000 }
gfCNCPoint1[8829] = {X 82.4647, Y 15.6039, Z -1.3333, A 0.000, B 0.000, C 0.000 }
gfCNCPoint1[8830] = {X 81.9836, Y 14.8119, Z -1.3333, A 0.000, B 0.000, C 0.000 }
gfCNCPoint1[8831] = {X 81.6825, Y 13.9354, Z -1.3333, A 0.000, B 0.000, C 0.000 }
gfCNCPoint1[8832] = {X 81.5752, Y 13.0150, Z -1.3333, A 0.000, B 0.000, C 0.000 }
gfCNCPoint1[8833] = {X 81.5751, Y 12.1868, Z -1.3333, A 0.000, B 0.000, C 0.000 }
gfCNCPoint1[8834] = {X 81.6834, Y 11.2255, Z -1.3333, A 0.000, B 0.000, C 0.000 }
gfCNCPoint1[8835] = {X 82.0029, Y 10.3125, Z -1.3333, A 0.000, B 0.000, C 0.000 }
gfCNCPoint1[8836] = {X 82.5176, Y 9.4933, Z -1.3333, A 0.000, B 0.000, C 0.000 }
gfCNCPoint1[8837] = {X 83.2016, Y 8.8093, Z -1.3333, A 0.000, B 0.000, C 0.000 }
gfCNCPoint1[8838] = {X 84.0207, Y 8.2946, Z -1.3333, A 0.000, B 0.000, C 0.000 }
gfCNCPoint1[8839] = {X 84.9338, Y 7.9751, Z -1.3333, A 0.000, B 0.000, C 0.000 }
gfCNCPoint1[8840] = {X 85.8951, Y 7.8668, Z -1.3333, A 0.000, B 0.000, C 0.000 }
gfCNCPoint1[8841] = {X 94.0497, Y 7.8668, Z -1.3333, A 0.000, B 0.000, C 0.000 }
gfCNCPoint1[8842] = {X 95.0110, Y 7.9751, Z -1.3333, A 0.000, B 0.000, C 0.000 }
gfCNCPoint1[8843] = {X 95.9240, Y 8.2946, Z -1.3333, A 0.000, B 0.000, C 0.000 }
gfCNCPoint1[8844] = {X 96.7431, Y 8.8093, Z -1.3333, A 0.000, B 0.000, C 0.000 }
gfCNCPoint1[8845] = {X 97.4272, Y 9.4933, Z -1.3333, A 0.000, B 0.000, C 0.000 }
gfCNCPoint1[8846] = {X 97.9419, Y 10.3124, Z -1.3333, A 0.000, B 0.000, C 0.000 }
gfCNCPoint1[8847] = {X 98.2614, Y 11.2255, Z -1.3333, A 0.000, B 0.000, C 0.000 }
gfCNCPoint1[8848] = {X 98.3697, Y 12.1868, Z -1.3333, A 0.000, B 0.000, C 0.000 }
gfCNCPoint1[8849] = {X 98.3697, Y 12.9781, Z -1.3333, A 0.000, B 0.000, C 0.000 }
gfCNCPoint1[8850] = {X 98.2966, Y 13.7685, Z -1.3333, A 0.000, B 0.000, C 0.000 }
gfCNCPoint1[8851] = {X 98.0802, Y 14.5321, Z -1.3333, A 0.000, B 0.000, C 0.000 }
gfCNCPoint1[8852] = {X 97.7277, Y 15.2433, Z -1.3333, A 0.000, B 0.000, C 0.000 }
gfCNCPoint1[8853] = {X 101.8783, Y 25.5307, Z -1.3333, A 0.000, B 0.000, C 0.000 }
gfCNCPoint1[8854] = {X 106.0169, Y 15.2222, Z -1.3333, A 0.000, B 0.000, C 0.000 }
gfCNCPoint1[8855] = {X 105.6763, Y 14.5291, Z -1.3333, A 0.000, B 0.000, C 0.000 }
gfCNCPoint1[8856] = {X 105.4646, Y 13.7864, Z -1.3333, A 0.000, B 0.000, C 0.000 }
gfCNCPoint1[8857] = {X 105.3885, Y 13.0179, Z -1.3333, A 0.000, B 0.000, C 0.000 }
gfCNCPoint1[8858] = {X 105.3883, Y 12.1868, Z -1.3333, A 0.000, B 0.000, C 0.000 }
gfCNCPoint1[8859] = {X 105.4966, Y 11.2255, Z -1.3333, A 0.000, B 0.000, C 0.000 }
gfCNCPoint1[8860] = {X 105.8161, Y 10.3124, Z -1.3333, A 0.000, B 0.000, C 0.000 }
gfCNCPoint1[8861] = {X 106.3308, Y 9.4933, Z -1.3333, A 0.000, B 0.000, C 0.000 }
gfCNCPoint1[8862] = {X 107.0148, Y 8.8093, Z -1.3333, A 0.000, B 0.000, C 0.000 }
gfCNCPoint1[8863] = {X 107.8339, Y 8.2946, Z -1.3333, A 0.000, B 0.000, C 0.000 }
gfCNCPoint1[8864] = {X 108.7470, Y 7.9751, Z -1.3333, A 0.000, B 0.000, C 0.000 }
gfCNCPoint1[8865] = {X 109.7083, Y 7.8668, Z -1.3333, A 0.000, B 0.000, C 0.000 }
gfCNCPoint1[8866] = {X 117.7916, Y 7.8668, Z -1.3333, A 0.000, B 0.000, C 0.000 }
gfCNCPoint1[8867] = {X 118.7529, Y 7.9751, Z -1.3333, A 0.000, B 0.000, C 0.000 }
gfCNCPoint1[8868] = {X 119.6660, Y 8.2946, Z -1.3333, A 0.000, B 0.000, C 0.000 }
gfCNCPoint1[8869] = {X 120.4851, Y 8.8093, Z -1.3333, A 0.000, B 0.000, C 0.000 }
gfCNCPoint1[8870] = {X 121.1691, Y 9.4933, Z -1.3333, A 0.000, B 0.000, C 0.000 }
gfCNCPoint1[8871] = {X 121.6838, Y 10.3124, Z -1.3333, A 0.000, B 0.000, C 0.000 }
gfCNCPoint1[8872] = {X 122.0033, Y 11.2255, Z -1.3333, A 0.000, B 0.000, C 0.000 }
gfCNCPoint1[8873] = {X 122.1116, Y 12.1868, Z -1.3333, A 0.000, B 0.000, C 0.000 }
gfCNCPoint1[8874] = {X 122.1116, Y 12.9781, Z -1.3333, A 0.000, B 0.000, C 0.000 }
gfCNCPoint1[8875] = {X 122.0103, Y 13.9081, Z -1.3333, A 0.000, B 0.000, C 0.000 }
gfCNCPoint1[8876] = {X 121.7111, Y 14.7945, Z -1.3333, A 0.000, B 0.000, C 0.000 }
gfCNCPoint1[8877] = {X 121.2282, Y 15.5957, Z -1.3333, A 0.000, B 0.000, C 0.000 }
gfCNCPoint1[8878] = {X 120.5841, Y 16.2741, Z -1.3333, A 0.000, B 0.000, C 0.000 }
gfCNCPoint1[8879] = {X 120.5828, Y 40.9135, Z -1.3333, A 0.000, B 0.000, C 0.000 }
gfCNCPoint1[8880] = {X 120.6215, Y 40.9448, Z -1.3333, A 0.000, B 0.000, C 0.000 }
gfCNCPoint1[8881] = {X 121.2452, Y 41.6136, Z -1.3333, A 0.000, B 0.000, C 0.000 }
gfCNCPoint1[8882] = {X 121.7141, Y 42.3987, Z -1.3333, A 0.000, B 0.000, C 0.000 }
gfCNCPoint1[8883] = {X 122.0072, Y 43.2649, Z -1.3333, A 0.000, B 0.000, C 0.000 }
gfCNCPoint1[8884] = {X 122.1114, Y 44.1734, Z -1.3333, A 0.000, B 0.000, C 0.000 }
gfCNCPoint1[8885] = {X 122.1116, Y 45.0000, Z -1.3333, A 0.000, B 0.000, C 0.000 }
gfCNCPoint1[8886] = {X 122.0033, Y 45.9613, Z -1.3333, A 0.000, B 0.000, C 0.000 }
gfCNCPoint1[8887] = {X 121.6838, Y 46.8744, Z -1.3333, A 0.000, B 0.000, C 0.000 }
gfCNCPoint1[8888] = {X 121.1691, Y 47.6935, Z -1.3333, A 0.000, B 0.000, C 0.000 }
gfCNCPoint1[8889] = {X 120.4851, Y 48.3775, Z -1.3333, A 0.000, B 0.000, C 0.000 }
gfCNCPoint1[8890] = {X 119.6660, Y 48.8922, Z -1.3333, A 0.000, B 0.000, C 0.000 }
gfCNCPoint1[8891] = {X 118.7529, Y 49.2117, Z -1.3333, A 0.000, B 0.000, C 0.000 }
gfCNCPoint1[8892] = {X 117.7916, Y 49.3200, Z -1.3333, A 0.000, B 0.000, C 0.000 }
gfCNCPoint1[8893] = {X 111.9185, Y 49.3200, Z -1.3333, A 0.000, B 0.000, C 0.000 }
gfCNCPoint1[8894] = {X 110.9619, Y 49.2128, Z -1.3333, A 0.000, B 0.000, C 0.000 }
gfCNCPoint1[8895] = {X 110.0529, Y 48.8964, Z -1.3333, A 0.000, B 0.000, C 0.000 }
gfCNCPoint1[8896] = {X 109.2365, Y 48.3866, Z -1.3333, A 0.000, B 0.000, C 0.000 }
gfCNCPoint1[8897] = {X 108.5532, Y 47.7087, Z -1.3333, A 0.000, B 0.000, C 0.000 }
gfCNCPoint1[8898] = {X 108.0369, Y 46.8963, Z -1.3333, A 0.000, B 0.000, C 0.000 }
gfCNCPoint1[8899] = {X 107.7134, Y 45.9898, Z -1.3333, A 0.000, B 0.000, C 0.000 }
gfCNCPoint1[8900] = {X 107.5986, Y 45.0341, Z -1.3333, A 0.000, B 0.000, C 0.000 }
gfCNCPoint1[8901] = {X 107.5985, Y 44.1795, Z -1.3333, A 0.000, B 0.000, C 0.000 }
gfCNCPoint1[8902] = {X 107.6344, Y 43.6351, Z -1.3333, A 0.000, B 0.000, C 0.000 }
gfCNCPoint1[8903] = {X 107.7414, Y 43.1000, Z -1.3333, A 0.000, B 0.000, C 0.000 }
gfCNCPoint1[8904] = {X 107.9074, Y 42.6088, Z -1.3333, A 0.000, B 0.000, C 0.000 }
gfCNCPoint1[8905] = {X 108.1334, Y 42.1422, Z -1.3333, A 0.000, B 0.000, C 0.000 }
gfCNCPoint1[8906] = {X 108.5855, Y 41.4674, Z -1.3333, A 0.000, B 0.000, C 0.000 }
gfCNCPoint1[8907] = {X 109.1273, Y 40.8622, Z -1.3333, A 0.000, B 0.000, C 0.000 }
gfCNCPoint1[8908] = {X 109.1272, Y 39.2929, Z -1.3333, A 0.000, B 0.000, C 0.000 }
gfCNCPoint1[8909] = {X 106.1118, Y 46.6615, Z -1.3333, A 0.000, B 0.000, C 0.000 }
gfCNCPoint1[8910] = {X 105.7417, Y 47.3611, Z -1.3333, A 0.000, B 0.000, C 0.000 }
gfCNCPoint1[8911] = {X 105.2502, Y 47.9815, Z -1.3333, A 0.000, B 0.000, C 0.000 }
gfCNCPoint1[8912] = {X 104.6538, Y 48.5018, Z -1.3333, A 0.000, B 0.000, C 0.000 }
gfCNCPoint1[8913] = {X 103.9724, Y 48.9046, Z -1.3333, A 0.000, B 0.000, C 0.000 }
gfCNCPoint1[8914] = {X 103.0287, Y 49.2242, Z -1.3333, A 0.000, B 0.000, C 0.000 }
gfCNCPoint1[8915] = {X 102.0368, Y 49.3191, Z -1.3333, A 0.000, B 0.000, C 0.000 }
gfCNCPoint1[8916] = {X 101.0496, Y 49.1842, Z -1.3333, A 0.000, B 0.000, C 0.000 }
gfCNCPoint1[8917] = {X 100.1195, Y 48.8268, Z -1.3333, A 0.000, B 0.000, C 0.000 }
gfCNCPoint1[8918] = {X 99.2961, Y 48.2657, Z -1.3333, A 0.000, B 0.000, C 0.000 }
gfCNCPoint1[8919] = {X 98.6231, Y 47.5309, Z -1.3333, A 0.000, B 0.000, C 0.000 }
gfCNCPoint1[8920] = {X 98.1363, Y 46.6615, Z -1.3333, A 0.000, B 0.000, C 0.000 }
gfCNCPoint1[8921] = {X 95.1297, Y 39.3085, Z -1.3333, A 0.000, B 0.000, C 0.000 }
gfCNCPoint1[8922] = {X 95.1299, Y 40.9056, Z -1.3333, A 0.000, B 0.000, C 0.000 }
gfCNCPoint1[8923] = {X 95.6605, Y 41.4499, Z -1.3333, A 0.000, B 0.000, C 0.000 }
gfCNCPoint1[8924] = {X 96.0896, Y 42.0773, Z -1.3333, A 0.000, B 0.000, C 0.000 }
gfCNCPoint1[8925] = {X 96.3307, Y 42.5752, Z -1.3333, A 0.000, B 0.000, C 0.000 }
gfCNCPoint1[8926] = {X 96.5076, Y 43.0994, Z -1.3333, A 0.000, B 0.000, C 0.000 }
gfCNCPoint1[8927] = {X 96.6182, Y 43.6480, Z -1.3333, A 0.000, B 0.000, C 0.000 }
gfCNCPoint1[8928] = {X 96.6585, Y 44.2062, Z -1.3333, A 0.000, B 0.000, C 0.000 }
gfCNCPoint1[8929] = {X 96.6583, Y 45.0415, Z -1.3333, A 0.000, B 0.000, C 0.000 }
gfCNCPoint1[8930] = {X 96.5422, Y 45.9960, Z -1.3333, A 0.000, B 0.000, C 0.000 }
gfCNCPoint1[8931] = {X 96.2178, Y 46.9011, Z -1.3333, A 0.000, B 0.000, C 0.000 }
gfCNCPoint1[8932] = {X 95.7012, Y 47.7120, Z -1.3333, A 0.000, B 0.000, C 0.000 }
gfCNCPoint1[8933] = {X 95.0181, Y 48.3886, Z -1.3333, A 0.000, B 0.000, C 0.000 }
gfCNCPoint1[8934] = {X 94.2022, Y 48.8973, Z -1.3333, A 0.000, B 0.000, C 0.000 }
gfCNCPoint1[8935] = {X 93.2940, Y 49.2130, Z -1.3333, A 0.000, B 0.000, C 0.000 }
gfCNCPoint1[8936] = {X 92.3385, Y 49.3200, Z -1.3333, A 0.000, B 0.000, C 0.000 }
gfCNCPoint1[8937] = {X 85.8951, Y 49.3200, Z -1.3333, A 0.000, B 0.000, C 0.000 }
gfCNCPoint1[8938] = {X 84.9387, Y 49.2128, Z -1.3333, A 0.000, B 0.000, C 0.000 }
gfCNCPoint1[8939] = {X 84.0297, Y 48.8965, Z -1.3333, A 0.000, B 0.000, C 0.000 }
gfCNCPoint1[8940] = {X 83.2134, Y 48.3869, Z -1.3333, A 0.000, B 0.000, C 0.000 }
gfCNCPoint1[8941] = {X 82.5301, Y 47.7091, Z -1.3333, A 0.000, B 0.000, C 0.000 }
gfCNCPoint1[8942] = {X 82.0138, Y 46.8970, Z -1.3333, A 0.000, B 0.000, C 0.000 }
gfCNCPoint1[8943] = {X 81.6902, Y 45.9906, Z -1.3333, A 0.000, B 0.000, C 0.000 }
gfCNCPoint1[8944] = {X 81.5752, Y 45.0351, Z -1.3333, A 0.000, B 0.000, C 0.000 }
gfCNCPoint1[8945] = {X 81.5751, Y 44.2067, Z -1.3333, A 0.000, B 0.000, C 0.000 }
gfCNCPoint1[8946] = {X 81.6811, Y 43.2777, Z -1.3333, A 0.000, B 0.000, C 0.000 }
gfCNCPoint1[8947] = {X 81.9818, Y 42.3923, Z -1.3333, A 0.000, B 0.000, C 0.000 }
gfCNCPoint1[8948] = {X 82.4634, Y 41.5908, Z -1.3333, A 0.000, B 0.000, C 0.000 }
gfCNCPoint1[8949] = {X 83.1040, Y 40.9096, Z -1.3333, A 0.000, B 0.000, C 0.000 }
gfCNCPoint1[8950] = {X 83.1039, Y 28.5924, Z -1.3333, A 0.000, B 0.000, C 0.000 }
gfCNCPoint1[8951] = {X 79.1039, Y 28.5924, Z -1.3333, A 0.000, B 0.000, C 0.000 }
gfCNCPoint1[8952] = {X 83.1839, Y 28.5924, Z -1.3333, A 0.000, B 0.000, C 0.000 }
gfCNCPoint1[8953] = {X 83.1837, Y 16.2378, Z -1.3333, A 0.000, B 0.000, C 0.000 }
gfCNCPoint1[8954] = {X 82.5452, Y 15.5772, Z -1.3333, A 0.000, B 0.000, C 0.000 }
gfCNCPoint1[8955] = {X 82.0639, Y 14.7946, Z -1.3333, A 0.000, B 0.000, C 0.000 }
gfCNCPoint1[8956] = {X 81.7626, Y 13.9267, Z -1.3333, A 0.000, B 0.000, C 0.000 }
gfCNCPoint1[8957] = {X 81.6552, Y 13.0143, Z -1.3333, A 0.000, B 0.000, C 0.000 }
gfCNCPoint1[8958] = {X 81.6551, Y 12.1868, Z -1.3333, A 0.000, B 0.000, C 0.000 }
gfCNCPoint1[8959] = {X 81.7614, Y 11.2433, Z -1.3333, A 0.000, B 0.000, C 0.000 }
gfCNCPoint1[8960] = {X 82.0750, Y 10.3472, Z -1.3333, A 0.000, B 0.000, C 0.000 }
gfCNCPoint1[8961] = {X 82.5801, Y 9.5432, Z -1.3333, A 0.000, B 0.000, C 0.000 }
gfCNCPoint1[8962] = {X 83.2515, Y 8.8719, Z -1.3333, A 0.000, B 0.000, C 0.000 }
gfCNCPoint1[8963] = {X 84.0554, Y 8.3667, Z -1.3333, A 0.000, B 0.000, C 0.000 }
gfCNCPoint1[8964] = {X 84.9516, Y 8.0531, Z -1.3333, A 0.000, B 0.000, C 0.000 }
gfCNCPoint1[8965] = {X 85.8951, Y 7.9468, Z -1.3333, A 0.000, B 0.000, C 0.000 }
gfCNCPoint1[8966] = {X 94.0497, Y 7.9468, Z -1.3333, A 0.000, B 0.000, C 0.000 }
gfCNCPoint1[8967] = {X 94.9932, Y 8.0531, Z -1.3333, A 0.000, B 0.000, C 0.000 }
gfCNCPoint1[8968] = {X 95.8893, Y 8.3667, Z -1.3333, A 0.000, B 0.000, C 0.000 }
gfCNCPoint1[8969] = {X 96.6933, Y 8.8718, Z -1.3333, A 0.000, B 0.000, C 0.000 }
gfCNCPoint1[8970] = {X 97.3646, Y 9.5432, Z -1.3333, A 0.000, B 0.000, C 0.000 }
gfCNCPoint1[8971] = {X 97.8698, Y 10.3471, Z -1.3333, A 0.000, B 0.000, C 0.000 }
gfCNCPoint1[8972] = {X 98.1834, Y 11.2433, Z -1.3333, A 0.000, B 0.000, C 0.000 }
gfCNCPoint1[8973] = {X 98.2897, Y 12.1868, Z -1.3333, A 0.000, B 0.000, C 0.000 }
gfCNCPoint1[8974] = {X 98.2897, Y 12.9781, Z -1.3333, A 0.000, B 0.000, C 0.000 }
gfCNCPoint1[8975] = {X 98.2155, Y 13.7670, Z -1.3333, A 0.000, B 0.000, C 0.000 }
gfCNCPoint1[8976] = {X 97.9958, Y 14.5283, Z -1.3333, A 0.000, B 0.000, C 0.000 }
gfCNCPoint1[8977] = {X 97.6383, Y 15.2355, Z -1.3333, A 0.000, B 0.000, C 0.000 }
gfCNCPoint1[8978] = {X 101.8782, Y 25.7443, Z -1.3333, A 0.000, B 0.000, C 0.000 }
gfCNCPoint1[8979] = {X 101.9525, Y 25.5605, Z -1.3333, A 0.000, B 0.000, C 0.000 }
gfCNCPoint1[8980] = {X 106.1062, Y 15.2146, Z -1.3333, A 0.000, B 0.000, C 0.000 }
gfCNCPoint1[8981] = {X 105.7606, Y 14.5252, Z -1.3333, A 0.000, B 0.000, C 0.000 }
gfCNCPoint1[8982] = {X 105.5457, Y 13.7845, Z -1.3333, A 0.000, B 0.000, C 0.000 }
gfCNCPoint1[8983] = {X 105.4685, Y 13.0172, Z -1.3333, A 0.000, B 0.000, C 0.000 }
gfCNCPoint1[8984] = {X 105.4683, Y 12.1868, Z -1.3333, A 0.000, B 0.000, C 0.000 }
gfCNCPoint1[8985] = {X 105.5746, Y 11.2433, Z -1.3333, A 0.000, B 0.000, C 0.000 }
gfCNCPoint1[8986] = {X 105.8882, Y 10.3471, Z -1.3333, A 0.000, B 0.000, C 0.000 }
gfCNCPoint1[8987] = {X 106.3933, Y 9.5432, Z -1.3333, A 0.000, B 0.000, C 0.000 }
gfCNCPoint1[8988] = {X 107.0647, Y 8.8718, Z -1.3333, A 0.000, B 0.000, C 0.000 }
gfCNCPoint1[8989] = {X 107.8686, Y 8.3667, Z -1.3333, A 0.000, B 0.000, C 0.000 }
gfCNCPoint1[8990] = {X 108.7648, Y 8.0531, Z -1.3333, A 0.000, B 0.000, C 0.000 }
gfCNCPoint1[8991] = {X 109.7083, Y 7.9468, Z -1.3333, A 0.000, B 0.000, C 0.000 }
gfCNCPoint1[8992] = {X 117.7916, Y 7.9468, Z -1.3333, A 0.000, B 0.000, C 0.000 }
gfCNCPoint1[8993] = {X 118.7351, Y 8.0531, Z -1.3333, A 0.000, B 0.000, C 0.000 }
gfCNCPoint1[8994] = {X 119.6312, Y 8.3667, Z -1.3333, A 0.000, B 0.000, C 0.000 }
gfCNCPoint1[8995] = {X 120.4352, Y 8.8718, Z -1.3333, A 0.000, B 0.000, C 0.000 }
gfCNCPoint1[8996] = {X 121.1065, Y 9.5432, Z -1.3333, A 0.000, B 0.000, C 0.000 }
gfCNCPoint1[8997] = {X 121.6117, Y 10.3471, Z -1.3333, A 0.000, B 0.000, C 0.000 }
gfCNCPoint1[8998] = {X 121.9253, Y 11.2433, Z -1.3333, A 0.000, B 0.000, C 0.000 }
gfCNCPoint1[8999] = {X 122.0316, Y 12.1868, Z -1.3333, A 0.000, B 0.000, C 0.000 }
gfCNCPoint1[9000] = {X 122.0316, Y 12.9781, Z -1.3333, A 0.000, B 0.000, C 0.000 }
gfCNCPoint1[9001] = {X 121.9301, Y 13.8999, Z -1.3333, A 0.000, B 0.000, C 0.000 }
gfCNCPoint1[9002] = {X 121.6307, Y 14.7776, Z -1.3333, A 0.000, B 0.000, C 0.000 }
gfCNCPoint1[9003] = {X 121.1477, Y 15.5692, Z -1.3333, A 0.000, B 0.000, C 0.000 }
gfCNCPoint1[9004] = {X 120.5041, Y 16.2368, Z -1.3333, A 0.000, B 0.000, C 0.000 }
gfCNCPoint1[9005] = {X 120.5028, Y 40.9518, Z -1.3333, A 0.000, B 0.000, C 0.000 }
gfCNCPoint1[9006] = {X 120.5701, Y 41.0061, Z -1.3333, A 0.000, B 0.000, C 0.000 }
gfCNCPoint1[9007] = {X 121.1818, Y 41.6625, Z -1.3333, A 0.000, B 0.000, C 0.000 }
gfCNCPoint1[9008] = {X 121.6417, Y 42.4328, Z -1.3333, A 0.000, B 0.000, C 0.000 }
gfCNCPoint1[9009] = {X 121.9292, Y 43.2827, Z -1.3333, A 0.000, B 0.000, C 0.000 }
gfCNCPoint1[9010] = {X 122.0314, Y 44.1740, Z -1.3333, A 0.000, B 0.000, C 0.000 }
gfCNCPoint1[9011] = {X 122.0316, Y 45.0000, Z -1.3333, A 0.000, B 0.000, C 0.000 }
gfCNCPoint1[9012] = {X 121.9253, Y 45.9435, Z -1.3333, A 0.000, B 0.000, C 0.000 }
gfCNCPoint1[9013] = {X 121.6117, Y 46.8397, Z -1.3333, A 0.000, B 0.000, C 0.000 }
gfCNCPoint1[9014] = {X 121.1065, Y 47.6436, Z -1.3333, A 0.000, B 0.000, C 0.000 }
gfCNCPoint1[9015] = {X 120.4352, Y 48.3150, Z -1.3333, A 0.000, B 0.000, C 0.000 }
gfCNCPoint1[9016] = {X 119.6312, Y 48.8201, Z -1.3333, A 0.000, B 0.000, C 0.000 }
gfCNCPoint1[9017] = {X 118.7351, Y 49.1337, Z -1.3333, A 0.000, B 0.000, C 0.000 }
gfCNCPoint1[9018] = {X 117.7916, Y 49.2400, Z -1.3333, A 0.000, B 0.000, C 0.000 }
gfCNCPoint1[9019] = {X 111.9185, Y 49.2400, Z -1.3333, A 0.000, B 0.000, C 0.000 }
gfCNCPoint1[9020] = {X 110.9797, Y 49.1348, Z -1.3333, A 0.000, B 0.000, C 0.000 }
gfCNCPoint1[9021] = {X 110.0874, Y 48.8242, Z -1.3333, A 0.000, B 0.000, C 0.000 }
gfCNCPoint1[9022] = {X 109.2861, Y 48.3239, Z -1.3333, A 0.000, B 0.000, C 0.000 }
gfCNCPoint1[9023] = {X 108.6155, Y 47.6585, Z -1.3333, A 0.000, B 0.000, C 0.000 }
gfCNCPoint1[9024] = {X 108.1088, Y 46.8612, Z -1.3333, A 0.000, B 0.000, C 0.000 }
gfCNCPoint1[9025] = {X 107.7913, Y 45.9714, Z -1.3333, A 0.000, B 0.000, C 0.000 }
gfCNCPoint1[9026] = {X 107.6786, Y 45.0335, Z -1.3333, A 0.000, B 0.000, C 0.000 }
gfCNCPoint1[9027] = {X 107.6785, Y 44.1795, Z -1.3333, A 0.000, B 0.000, C 0.000 }
gfCNCPoint1[9028] = {X 107.7137, Y 43.6456, Z -1.3333, A 0.000, B 0.000, C 0.000 }
gfCNCPoint1[9029] = {X 107.8187, Y 43.1209, Z -1.3333, A 0.000, B 0.000, C 0.000 }
gfCNCPoint1[9030] = {X 107.9815, Y 42.6391, Z -1.3333, A 0.000, B 0.000, C 0.000 }
gfCNCPoint1[9031] = {X 108.2031, Y 42.1815, Z -1.3333, A 0.000, B 0.000, C 0.000 }
gfCNCPoint1[9032] = {X 108.6592, Y 41.5029, Z -1.3333, A 0.000, B 0.000, C 0.000 }
gfCNCPoint1[9033] = {X 109.2073, Y 40.8962, Z -1.3333, A 0.000, B 0.000, C 0.000 }
gfCNCPoint1[9034] = {X 109.2071, Y 39.1629, Z -1.3333, A 0.000, B 0.000, C 0.000 }
gfCNCPoint1[9035] = {X 109.0939, Y 39.1629, Z -1.3333, A 0.000, B 0.000, C 0.000 }
gfCNCPoint1[9036] = {X 106.0379, Y 46.6307, Z -1.3333, A 0.000, B 0.000, C 0.000 }
gfCNCPoint1[9037] = {X 105.6747, Y 47.3174, Z -1.3333, A 0.000, B 0.000, C 0.000 }
gfCNCPoint1[9038] = {X 105.1923, Y 47.9263, Z -1.3333, A 0.000, B 0.000, C 0.000 }
gfCNCPoint1[9039] = {X 104.6069, Y 48.4370, Z -1.3333, A 0.000, B 0.000, C 0.000 }
gfCNCPoint1[9040] = {X 103.9382, Y 48.8323, Z -1.3333, A 0.000, B 0.000, C 0.000 }
gfCNCPoint1[9041] = {X 103.0119, Y 49.1460, Z -1.3333, A 0.000, B 0.000, C 0.000 }
gfCNCPoint1[9042] = {X 102.0384, Y 49.2391, Z -1.3333, A 0.000, B 0.000, C 0.000 }
gfCNCPoint1[9043] = {X 101.0695, Y 49.1068, Z -1.3333, A 0.000, B 0.000, C 0.000 }
gfCNCPoint1[9044] = {X 100.1566, Y 48.7559, Z -1.3333, A 0.000, B 0.000, C 0.000 }
gfCNCPoint1[9045] = {X 99.3484, Y 48.2052, Z -1.3333, A 0.000, B 0.000, C 0.000 }
gfCNCPoint1[9046] = {X 98.6879, Y 47.4840, Z -1.3333, A 0.000, B 0.000, C 0.000 }
gfCNCPoint1[9047] = {X 98.2102, Y 46.6307, Z -1.3333, A 0.000, B 0.000, C 0.000 }
gfCNCPoint1[9048] = {X 95.0497, Y 38.9014, Z -1.3333, A 0.000, B 0.000, C 0.000 }
gfCNCPoint1[9049] = {X 95.0499, Y 40.9425, Z -1.3333, A 0.000, B 0.000, C 0.000 }
gfCNCPoint1[9050] = {X 95.5870, Y 41.4865, Z -1.3333, A 0.000, B 0.000, C 0.000 }
gfCNCPoint1[9051] = {X 96.0200, Y 42.1166, Z -1.3333, A 0.000, B 0.000, C 0.000 }
gfCNCPoint1[9052] = {X 96.2567, Y 42.6055, Z -1.3333, A 0.000, B 0.000, C 0.000 }
gfCNCPoint1[9053] = {X 96.4303, Y 43.1201, Z -1.3333, A 0.000, B 0.000, C 0.000 }
gfCNCPoint1[9054] = {X 96.5390, Y 43.6588, Z -1.3333, A 0.000, B 0.000, C 0.000 }
gfCNCPoint1[9055] = {X 96.5785, Y 44.2069, Z -1.3333, A 0.000, B 0.000, C 0.000 }
gfCNCPoint1[9056] = {X 96.5783, Y 45.0408, Z -1.3333, A 0.000, B 0.000, C 0.000 }
gfCNCPoint1[9057] = {X 96.4643, Y 45.9775, Z -1.3333, A 0.000, B 0.000, C 0.000 }
gfCNCPoint1[9058] = {X 96.1459, Y 46.8659, Z -1.3333, A 0.000, B 0.000, C 0.000 }
gfCNCPoint1[9059] = {X 95.6389, Y 47.6618, Z -1.3333, A 0.000, B 0.000, C 0.000 }
gfCNCPoint1[9060] = {X 94.9685, Y 48.3258, Z -1.3333, A 0.000, B 0.000, C 0.000 }
gfCNCPoint1[9061] = {X 94.1677, Y 48.8251, Z -1.3333, A 0.000, B 0.000, C 0.000 }
gfCNCPoint1[9062] = {X 93.2764, Y 49.1350, Z -1.3333, A 0.000, B 0.000, C 0.000 }
gfCNCPoint1[9063] = {X 92.3385, Y 49.2400, Z -1.3333, A 0.000, B 0.000, C 0.000 }
gfCNCPoint1[9064] = {X 85.8951, Y 49.2400, Z -1.3333, A 0.000, B 0.000, C 0.000 }
gfCNCPoint1[9065] = {X 84.9564, Y 49.1348, Z -1.3333, A 0.000, B 0.000, C 0.000 }
gfCNCPoint1[9066] = {X 84.0643, Y 48.8244, Z -1.3333, A 0.000, B 0.000, C 0.000 }
gfCNCPoint1[9067] = {X 83.2631, Y 48.3242, Z -1.3333, A 0.000, B 0.000, C 0.000 }
gfCNCPoint1[9068] = {X 82.5924, Y 47.6590, Z -1.3333, A 0.000, B 0.000, C 0.000 }
gfCNCPoint1[9069] = {X 82.0857, Y 46.8618, Z -1.3333, A 0.000, B 0.000, C 0.000 }
gfCNCPoint1[9070] = {X 81.7681, Y 45.9723, Z -1.3333, A 0.000, B 0.000, C 0.000 }
gfCNCPoint1[9071] = {X 81.6552, Y 45.0345, Z -1.3333, A 0.000, B 0.000, C 0.000 }
gfCNCPoint1[9072] = {X 81.6551, Y 44.2073, Z -1.3333, A 0.000, B 0.000, C 0.000 }
gfCNCPoint1[9073] = {X 81.7612, Y 43.2863, Z -1.3333, A 0.000, B 0.000, C 0.000 }
gfCNCPoint1[9074] = {X 82.0621, Y 42.4093, Z -1.3333, A 0.000, B 0.000, C 0.000 }
gfCNCPoint1[9075] = {X 82.5438, Y 41.6172, Z -1.3333, A 0.000, B 0.000, C 0.000 }
gfCNCPoint1[9076] = {X 83.1840, Y 40.9466, Z -1.3333, A 0.000, B 0.000, C 0.000 }
gfCNCPoint1[9077] = {X 83.1839, Y 28.5924, Z -1.3333, A 0.000, B 0.000, C 0.000 }
gfCNCPoint1[9078] = {X 79.1839, Y 28.5924, Z -1.3333, A 0.000, B 0.000, C 0.000 }
gfCNCPoint1[9079] = {X 83.2639, Y 28.5924, Z -1.3333, A 0.000, B 0.000, C 0.000 }
gfCNCPoint1[9080] = {X 83.2637, Y 16.2001, Z -1.3333, A 0.000, B 0.000, C 0.000 }
gfCNCPoint1[9081] = {X 82.6257, Y 15.5503, Z -1.3333, A 0.000, B 0.000, C 0.000 }
gfCNCPoint1[9082] = {X 82.1443, Y 14.7772, Z -1.3333, A 0.000, B 0.000, C 0.000 }
gfCNCPoint1[9083] = {X 81.8426, Y 13.9179, Z -1.3333, A 0.000, B 0.000, C 0.000 }
gfCNCPoint1[9084] = {X 81.7352, Y 13.0136, Z -1.3333, A 0.000, B 0.000, C 0.000 }
gfCNCPoint1[9085] = {X 81.7351, Y 12.1868, Z -1.3333, A 0.000, B 0.000, C 0.000 }
gfCNCPoint1[9086] = {X 81.8394, Y 11.2611, Z -1.3333, A 0.000, B 0.000, C 0.000 }
gfCNCPoint1[9087] = {X 82.1470, Y 10.3819, Z -1.3333, A 0.000, B 0.000, C 0.000 }
gfCNCPoint1[9088] = {X 82.6427, Y 9.5931, Z -1.3333, A 0.000, B 0.000, C 0.000 }
gfCNCPoint1[9089] = {X 83.3014, Y 8.9344, Z -1.3333, A 0.000, B 0.000, C 0.000 }
gfCNCPoint1[9090] = {X 84.0901, Y 8.4388, Z -1.3333, A 0.000, B 0.000, C 0.000 }
gfCNCPoint1[9091] = {X 84.9694, Y 8.1311, Z -1.3333, A 0.000, B 0.000, C 0.000 }
gfCNCPoint1[9092] = {X 85.8951, Y 8.0268, Z -1.3333, A 0.000, B 0.000, C 0.000 }
gfCNCPoint1[9093] = {X 94.0497, Y 8.0268, Z -1.3333, A 0.000, B 0.000, C 0.000 }
gfCNCPoint1[9094] = {X 94.9754, Y 8.1311, Z -1.3333, A 0.000, B 0.000, C 0.000 }
gfCNCPoint1[9095] = {X 95.8546, Y 8.4388, Z -1.3333, A 0.000, B 0.000, C 0.000 }
gfCNCPoint1[9096] = {X 96.6434, Y 8.9344, Z -1.3333, A 0.000, B 0.000, C 0.000 }
gfCNCPoint1[9097] = {X 97.3021, Y 9.5931, Z -1.3333, A 0.000, B 0.000, C 0.000 }
gfCNCPoint1[9098] = {X 97.7977, Y 10.3819, Z -1.3333, A 0.000, B 0.000, C 0.000 }
gfCNCPoint1[9099] = {X 98.1054, Y 11.2611, Z -1.3333, A 0.000, B 0.000, C 0.000 }
gfCNCPoint1[9100] = {X 98.2097, Y 12.1868, Z -1.3333, A 0.000, B 0.000, C 0.000 }
gfCNCPoint1[9101] = {X 98.2097, Y 12.9781, Z -1.3333, A 0.000, B 0.000, C 0.000 }
gfCNCPoint1[9102] = {X 98.1343, Y 13.7663, Z -1.3333, A 0.000, B 0.000, C 0.000 }
gfCNCPoint1[9103] = {X 97.9109, Y 14.5260, Z -1.3333, A 0.000, B 0.000, C 0.000 }
gfCNCPoint1[9104] = {X 97.5477, Y 15.2295, Z -1.3333, A 0.000, B 0.000, C 0.000 }
gfCNCPoint1[9105] = {X 101.8776, Y 25.9567, Z -1.3333, A 0.000, B 0.000, C 0.000 }
gfCNCPoint1[9106] = {X 101.9792, Y 25.7088, Z -1.3333, A 0.000, B 0.000, C 0.000 }
gfCNCPoint1[9107] = {X 106.1956, Y 15.2066, Z -1.3333, A 0.000, B 0.000, C 0.000 }
gfCNCPoint1[9108] = {X 105.8450, Y 14.5210, Z -1.3333, A 0.000, B 0.000, C 0.000 }
gfCNCPoint1[9109] = {X 105.6268, Y 13.7825, Z -1.3333, A 0.000, B 0.000, C 0.000 }
gfCNCPoint1[9110] = {X 105.5485, Y 13.0164, Z -1.3333, A 0.000, B 0.000, C 0.000 }
gfCNCPoint1[9111] = {X 105.5483, Y 12.1868, Z -1.3333, A 0.000, B 0.000, C 0.000 }
gfCNCPoint1[9112] = {X 105.6526, Y 11.2611, Z -1.3333, A 0.000, B 0.000, C 0.000 }
gfCNCPoint1[9113] = {X 105.9602, Y 10.3819, Z -1.3333, A 0.000, B 0.000, C 0.000 }
gfCNCPoint1[9114] = {X 106.4559, Y 9.5931, Z -1.3333, A 0.000, B 0.000, C 0.000 }
gfCNCPoint1[9115] = {X 107.1146, Y 8.9344, Z -1.3333, A 0.000, B 0.000, C 0.000 }
gfCNCPoint1[9116] = {X 107.9033, Y 8.4388, Z -1.3333, A 0.000, B 0.000, C 0.000 }
gfCNCPoint1[9117] = {X 108.7826, Y 8.1311, Z -1.3333, A 0.000, B 0.000, C 0.000 }
gfCNCPoint1[9118] = {X 109.7083, Y 8.0268, Z -1.3333, A 0.000, B 0.000, C 0.000 }
gfCNCPoint1[9119] = {X 117.7916, Y 8.0268, Z -1.3333, A 0.000, B 0.000, C 0.000 }
gfCNCPoint1[9120] = {X 118.7173, Y 8.1311, Z -1.3333, A 0.000, B 0.000, C 0.000 }
gfCNCPoint1[9121] = {X 119.5965, Y 8.4388, Z -1.3333, A 0.000, B 0.000, C 0.000 }
gfCNCPoint1[9122] = {X 120.3853, Y 8.9344, Z -1.3333, A 0.000, B 0.000, C 0.000 }
gfCNCPoint1[9123] = {X 121.0440, Y 9.5931, Z -1.3333, A 0.000, B 0.000, C 0.000 }
gfCNCPoint1[9124] = {X 121.5396, Y 10.3819, Z -1.3333, A 0.000, B 0.000, C 0.000 }
gfCNCPoint1[9125] = {X 121.8473, Y 11.2611, Z -1.3333, A 0.000, B 0.000, C 0.000 }
gfCNCPoint1[9126] = {X 121.9516, Y 12.1868, Z -1.3333, A 0.000, B 0.000, C 0.000 }
gfCNCPoint1[9127] = {X 121.9516, Y 12.9781, Z -1.3333, A 0.000, B 0.000, C 0.000 }
gfCNCPoint1[9128] = {X 121.8500, Y 13.8916, Z -1.3333, A 0.000, B 0.000, C 0.000 }
gfCNCPoint1[9129] = {X 121.5503, Y 14.7605, Z -1.3333, A 0.000, B 0.000, C 0.000 }
gfCNCPoint1[9130] = {X 121.0672, Y 15.5424, Z -1.3333, A 0.000, B 0.000, C 0.000 }
gfCNCPoint1[9131] = {X 120.4241, Y 16.1991, Z -1.3333, A 0.000, B 0.000, C 0.000 }
gfCNCPoint1[9132] = {X 120.4228, Y 40.9900, Z -1.3333, A 0.000, B 0.000, C 0.000 }
gfCNCPoint1[9133] = {X 120.5188, Y 41.0675, Z -1.3333, A 0.000, B 0.000, C 0.000 }
gfCNCPoint1[9134] = {X 121.1185, Y 41.7113, Z -1.3333, A 0.000, B 0.000, C 0.000 }
gfCNCPoint1[9135] = {X 121.5694, Y 42.4670, Z -1.3333, A 0.000, B 0.000, C 0.000 }
gfCNCPoint1[9136] = {X 121.8512, Y 43.3005, Z -1.3333, A 0.000, B 0.000, C 0.000 }
gfCNCPoint1[9137] = {X 121.9514, Y 44.1747, Z -1.3333, A 0.000, B 0.000, C 0.000 }
gfCNCPoint1[9138] = {X 121.9516, Y 45.0000, Z -1.3333, A 0.000, B 0.000, C 0.000 }
gfCNCPoint1[9139] = {X 121.8473, Y 45.9257, Z -1.3333, A 0.000, B 0.000, C 0.000 }
gfCNCPoint1[9140] = {X 121.5396, Y 46.8050, Z -1.3333, A 0.000, B 0.000, C 0.000 }
gfCNCPoint1[9141] = {X 121.0440, Y 47.5937, Z -1.3333, A 0.000, B 0.000, C 0.000 }
gfCNCPoint1[9142] = {X 120.3853, Y 48.2524, Z -1.3333, A 0.000, B 0.000, C 0.000 }
gfCNCPoint1[9143] = {X 119.5965, Y 48.7480, Z -1.3333, A 0.000, B 0.000, C 0.000 }
gfCNCPoint1[9144] = {X 118.7173, Y 49.0557, Z -1.3333, A 0.000, B 0.000, C 0.000 }
gfCNCPoint1[9145] = {X 117.7916, Y 49.1600, Z -1.3333, A 0.000, B 0.000, C 0.000 }
gfCNCPoint1[9146] = {X 111.9185, Y 49.1600, Z -1.3333, A 0.000, B 0.000, C 0.000 }
gfCNCPoint1[9147] = {X 110.9974, Y 49.0567, Z -1.3333, A 0.000, B 0.000, C 0.000 }
gfCNCPoint1[9148] = {X 110.1220, Y 48.7521, Z -1.3333, A 0.000, B 0.000, C 0.000 }
gfCNCPoint1[9149] = {X 109.3358, Y 48.2612, Z -1.3333, A 0.000, B 0.000, C 0.000 }
gfCNCPoint1[9150] = {X 108.6778, Y 47.6084, Z -1.3333, A 0.000, B 0.000, C 0.000 }
gfCNCPoint1[9151] = {X 108.1807, Y 46.8261, Z -1.3333, A 0.000, B 0.000, C 0.000 }
gfCNCPoint1[9152] = {X 107.8691, Y 45.9531, Z -1.3333, A 0.000, B 0.000, C 0.000 }
gfCNCPoint1[9153] = {X 107.7586, Y 45.0328, Z -1.3333, A 0.000, B 0.000, C 0.000 }
gfCNCPoint1[9154] = {X 107.7585, Y 44.1795, Z -1.3333, A 0.000, B 0.000, C 0.000 }
gfCNCPoint1[9155] = {X 107.7930, Y 43.6561, Z -1.3333, A 0.000, B 0.000, C 0.000 }
gfCNCPoint1[9156] = {X 107.8959, Y 43.1417, Z -1.3333, A 0.000, B 0.000, C 0.000 }
gfCNCPoint1[9157] = {X 108.0555, Y 42.6694, Z -1.3333, A 0.000, B 0.000, C 0.000 }
gfCNCPoint1[9158] = {X 108.2728, Y 42.2208, Z -1.3333, A 0.000, B 0.000, C 0.000 }
gfCNCPoint1[9159] = {X 108.7329, Y 41.5386, Z -1.3333, A 0.000, B 0.000, C 0.000 }
gfCNCPoint1[9160] = {X 109.2873, Y 40.9305, Z -1.3333, A 0.000, B 0.000, C 0.000 }
gfCNCPoint1[9161] = {X 109.2871, Y 39.0829, Z -1.3333, A 0.000, B 0.000, C 0.000 }
gfCNCPoint1[9162] = {X 109.0402, Y 39.0829, Z -1.3333, A 0.000, B 0.000, C 0.000 }
gfCNCPoint1[9163] = {X 105.9641, Y 46.5999, Z -1.3333, A 0.000, B 0.000, C 0.000 }
gfCNCPoint1[9164] = {X 105.6077, Y 47.2737, Z -1.3333, A 0.000, B 0.000, C 0.000 }
gfCNCPoint1[9165] = {X 105.1344, Y 47.8711, Z -1.3333, A 0.000, B 0.000, C 0.000 }
gfCNCPoint1[9166] = {X 104.5601, Y 48.3721, Z -1.3333, A 0.000, B 0.000, C 0.000 }
gfCNCPoint1[9167] = {X 103.9040, Y 48.7600, Z -1.3333, A 0.000, B 0.000, C 0.000 }
gfCNCPoint1[9168] = {X 102.9952, Y 49.0678, Z -1.3333, A 0.000, B 0.000, C 0.000 }
gfCNCPoint1[9169] = {X 102.0400, Y 49.1592, Z -1.3333, A 0.000, B 0.000, C 0.000 }
gfCNCPoint1[9170] = {X 101.0894, Y 49.0293, Z -1.3333, A 0.000, B 0.000, C 0.000 }
gfCNCPoint1[9171] = {X 100.1937, Y 48.6850, Z -1.3333, A 0.000, B 0.000, C 0.000 }
gfCNCPoint1[9172] = {X 99.4008, Y 48.1448, Z -1.3333, A 0.000, B 0.000, C 0.000 }
gfCNCPoint1[9173] = {X 98.7527, Y 47.4372, Z -1.3333, A 0.000, B 0.000, C 0.000 }
gfCNCPoint1[9174] = {X 98.2840, Y 46.5999, Z -1.3333, A 0.000, B 0.000, C 0.000 }
gfCNCPoint1[9175] = {X 94.9697, Y 38.4943, Z -1.3333, A 0.000, B 0.000, C 0.000 }
gfCNCPoint1[9176] = {X 94.9699, Y 40.9797, Z -1.3333, A 0.000, B 0.000, C 0.000 }
gfCNCPoint1[9177] = {X 95.5135, Y 41.5233, Z -1.3333, A 0.000, B 0.000, C 0.000 }
gfCNCPoint1[9178] = {X 95.9503, Y 42.1559, Z -1.3333, A 0.000, B 0.000, C 0.000 }
gfCNCPoint1[9179] = {X 96.1826, Y 42.6357, Z -1.3333, A 0.000, B 0.000, C 0.000 }
gfCNCPoint1[9180] = {X 96.3530, Y 43.1409, Z -1.3333, A 0.000, B 0.000, C 0.000 }
gfCNCPoint1[9181] = {X 96.4597, Y 43.6696, Z -1.3333, A 0.000, B 0.000, C 0.000 }
gfCNCPoint1[9182] = {X 96.4985, Y 44.2076, Z -1.3333, A 0.000, B 0.000, C 0.000 }
gfCNCPoint1[9183] = {X 96.4983, Y 45.0400, Z -1.3333, A 0.000, B 0.000, C 0.000 }
gfCNCPoint1[9184] = {X 96.3865, Y 45.9591, Z -1.3333, A 0.000, B 0.000, C 0.000 }
gfCNCPoint1[9185] = {X 96.0741, Y 46.8306, Z -1.3333, A 0.000, B 0.000, C 0.000 }
gfCNCPoint1[9186] = {X 95.5767, Y 47.6115, Z -1.3333, A 0.000, B 0.000, C 0.000 }
gfCNCPoint1[9187] = {X 94.9188, Y 48.2631, Z -1.3333, A 0.000, B 0.000, C 0.000 }
gfCNCPoint1[9188] = {X 94.1332, Y 48.7530, Z -1.3333, A 0.000, B 0.000, C 0.000 }
gfCNCPoint1[9189] = {X 93.2587, Y 49.0570, Z -1.3333, A 0.000, B 0.000, C 0.000 }
gfCNCPoint1[9190] = {X 92.3385, Y 49.1600, Z -1.3333, A 0.000, B 0.000, C 0.000 }
gfCNCPoint1[9191] = {X 85.8951, Y 49.1600, Z -1.3333, A 0.000, B 0.000, C 0.000 }
gfCNCPoint1[9192] = {X 84.9741, Y 49.0568, Z -1.3333, A 0.000, B 0.000, C 0.000 }
gfCNCPoint1[9193] = {X 84.0988, Y 48.7522, Z -1.3333, A 0.000, B 0.000, C 0.000 }
gfCNCPoint1[9194] = {X 83.3127, Y 48.2614, Z -1.3333, A 0.000, B 0.000, C 0.000 }
gfCNCPoint1[9195] = {X 82.6547, Y 47.6088, Z -1.3333, A 0.000, B 0.000, C 0.000 }
gfCNCPoint1[9196] = {X 82.1576, Y 46.8267, Z -1.3333, A 0.000, B 0.000, C 0.000 }
gfCNCPoint1[9197] = {X 81.8459, Y 45.9539, Z -1.3333, A 0.000, B 0.000, C 0.000 }
gfCNCPoint1[9198] = {X 81.7352, Y 45.0338, Z -1.3333, A 0.000, B 0.000, C 0.000 }
gfCNCPoint1[9199] = {X 81.7351, Y 44.2078, Z -1.3333, A 0.000, B 0.000, C 0.000 }
gfCNCPoint1[9200] = {X 81.8413, Y 43.2949, Z -1.3333, A 0.000, B 0.000, C 0.000 }
gfCNCPoint1[9201] = {X 82.1424, Y 42.4265, Z -1.3333, A 0.000, B 0.000, C 0.000 }
gfCNCPoint1[9202] = {X 82.6243, Y 41.6439, Z -1.3333, A 0.000, B 0.000, C 0.000 }
gfCNCPoint1[9203] = {X 83.2640, Y 40.9840, Z -1.3333, A 0.000, B 0.000, C 0.000 }
gfCNCPoint1[9204] = {X 83.2639, Y 28.5924, Z -1.3333, A 0.000, B 0.000, C 0.000 }
gfCNCPoint1[9205] = {X 79.2639, Y 28.5924, Z -1.3333, A 0.000, B 0.000, C 0.000 }
gfCNCPoint1[9206] = {X 83.3439, Y 28.5924, Z -1.3333, A 0.000, B 0.000, C 0.000 }
gfCNCPoint1[9207] = {X 83.3437, Y 16.1619, Z -1.3333, A 0.000, B 0.000, C 0.000 }
gfCNCPoint1[9208] = {X 82.7061, Y 15.5230, Z -1.3333, A 0.000, B 0.000, C 0.000 }
gfCNCPoint1[9209] = {X 82.2246, Y 14.7596, Z -1.3333, A 0.000, B 0.000, C 0.000 }
gfCNCPoint1[9210] = {X 81.9227, Y 13.9091, Z -1.3333, A 0.000, B 0.000, C 0.000 }
gfCNCPoint1[9211] = {X 81.8152, Y 13.0129, Z -1.3333, A 0.000, B 0.000, C 0.000 }
gfCNCPoint1[9212] = {X 81.8151, Y 12.1868, Z -1.3333, A 0.000, B 0.000, C 0.000 }
gfCNCPoint1[9213] = {X 81.9174, Y 11.2789, Z -1.3333, A 0.000, B 0.000, C 0.000 }
gfCNCPoint1[9214] = {X 82.2191, Y 10.4166, Z -1.3333, A 0.000, B 0.000, C 0.000 }
gfCNCPoint1[9215] = {X 82.7052, Y 9.6430, Z -1.3333, A 0.000, B 0.000, C 0.000 }
gfCNCPoint1[9216] = {X 83.3512, Y 8.9969, Z -1.3333, A 0.000, B 0.000, C 0.000 }
gfCNCPoint1[9217] = {X 84.1248, Y 8.5109, Z -1.3333, A 0.000, B 0.000, C 0.000 }
gfCNCPoint1[9218] = {X 84.9872, Y 8.2091, Z -1.3333, A 0.000, B 0.000, C 0.000 }
gfCNCPoint1[9219] = {X 85.8951, Y 8.1068, Z -1.3333, A 0.000, B 0.000, C 0.000 }
gfCNCPoint1[9220] = {X 94.0497, Y 8.1068, Z -1.3333, A 0.000, B 0.000, C 0.000 }
gfCNCPoint1[9221] = {X 94.9576, Y 8.2091, Z -1.3333, A 0.000, B 0.000, C 0.000 }
gfCNCPoint1[9222] = {X 95.8199, Y 8.5109, Z -1.3333, A 0.000, B 0.000, C 0.000 }
gfCNCPoint1[9223] = {X 96.5935, Y 8.9969, Z -1.3333, A 0.000, B 0.000, C 0.000 }
gfCNCPoint1[9224] = {X 97.2395, Y 9.6430, Z -1.3333, A 0.000, B 0.000, C 0.000 }
gfCNCPoint1[9225] = {X 97.7256, Y 10.4166, Z -1.3333, A 0.000, B 0.000, C 0.000 }
gfCNCPoint1[9226] = {X 98.0274, Y 11.2789, Z -1.3333, A 0.000, B 0.000, C 0.000 }
gfCNCPoint1[9227] = {X 98.1297, Y 12.1868, Z -1.3333, A 0.000, B 0.000, C 0.000 }
gfCNCPoint1[9228] = {X 98.1297, Y 12.9781, Z -1.3333, A 0.000, B 0.000, C 0.000 }
gfCNCPoint1[9229] = {X 98.0630, Y 13.7124, Z -1.3333, A 0.000, B 0.000, C 0.000 }
gfCNCPoint1[9230] = {X 97.8653, Y 14.4227, Z -1.3333, A 0.000, B 0.000, C 0.000 }
gfCNCPoint1[9231] = {X 97.5430, Y 15.0859, Z -1.3333, A 0.000, B 0.000, C 0.000 }
gfCNCPoint1[9232] = {X 97.4967, Y 15.1607, Z -1.3333, A 0.000, B 0.000, C 0.000 }
gfCNCPoint1[9233] = {X 97.4489, Y 15.2345, Z -1.3333, A 0.000, B 0.000, C 0.000 }
gfCNCPoint1[9234] = {X 97.4841, Y 15.2809, Z -1.3333, A 0.000, B 0.000, C 0.000 }
gfCNCPoint1[9235] = {X 101.8771, Y 26.1691, Z -1.3333, A 0.000, B 0.000, C 0.000 }
gfCNCPoint1[9236] = {X 102.0533, Y 25.7388, Z -1.3333, A 0.000, B 0.000, C 0.000 }
gfCNCPoint1[9237] = {X 106.2852, Y 15.1982, Z -1.3333, A 0.000, B 0.000, C 0.000 }
gfCNCPoint1[9238] = {X 106.2419, Y 15.1299, Z -1.3333, A 0.000, B 0.000, C 0.000 }
gfCNCPoint1[9239] = {X 106.1999, Y 15.0608, Z -1.3333, A 0.000, B 0.000, C 0.000 }
gfCNCPoint1[9240] = {X 105.8902, Y 14.4162, Z -1.3333, A 0.000, B 0.000, C 0.000 }
gfCNCPoint1[9241] = {X 105.6977, Y 13.7275, Z -1.3333, A 0.000, B 0.000, C 0.000 }
gfCNCPoint1[9242] = {X 105.6285, Y 13.0157, Z -1.3333, A 0.000, B 0.000, C 0.000 }
gfCNCPoint1[9243] = {X 105.6283, Y 12.1868, Z -1.3333, A 0.000, B 0.000, C 0.000 }
gfCNCPoint1[9244] = {X 105.7306, Y 11.2789, Z -1.3333, A 0.000, B 0.000, C 0.000 }
gfCNCPoint1[9245] = {X 106.0323, Y 10.4166, Z -1.3333, A 0.000, B 0.000, C 0.000 }
gfCNCPoint1[9246] = {X 106.5184, Y 9.6430, Z -1.3333, A 0.000, B 0.000, C 0.000 }
gfCNCPoint1[9247] = {X 107.1644, Y 8.9969, Z -1.3333, A 0.000, B 0.000, C 0.000 }
gfCNCPoint1[9248] = {X 107.9380, Y 8.5109, Z -1.3333, A 0.000, B 0.000, C 0.000 }
gfCNCPoint1[9249] = {X 108.8004, Y 8.2091, Z -1.3333, A 0.000, B 0.000, C 0.000 }
gfCNCPoint1[9250] = {X 109.7083, Y 8.1068, Z -1.3333, A 0.000, B 0.000, C 0.000 }
gfCNCPoint1[9251] = {X 117.7916, Y 8.1068, Z -1.3333, A 0.000, B 0.000, C 0.000 }
gfCNCPoint1[9252] = {X 118.6995, Y 8.2091, Z -1.3333, A 0.000, B 0.000, C 0.000 }
gfCNCPoint1[9253] = {X 119.5618, Y 8.5109, Z -1.3333, A 0.000, B 0.000, C 0.000 }
gfCNCPoint1[9254] = {X 120.3354, Y 8.9969, Z -1.3333, A 0.000, B 0.000, C 0.000 }
gfCNCPoint1[9255] = {X 120.9814, Y 9.6430, Z -1.3333, A 0.000, B 0.000, C 0.000 }
gfCNCPoint1[9256] = {X 121.4675, Y 10.4166, Z -1.3333, A 0.000, B 0.000, C 0.000 }
gfCNCPoint1[9257] = {X 121.7693, Y 11.2789, Z -1.3333, A 0.000, B 0.000, C 0.000 }
gfCNCPoint1[9258] = {X 121.8716, Y 12.1868, Z -1.3333, A 0.000, B 0.000, C 0.000 }
gfCNCPoint1[9259] = {X 121.8716, Y 12.9781, Z -1.3333, A 0.000, B 0.000, C 0.000 }
gfCNCPoint1[9260] = {X 121.7699, Y 13.8833, Z -1.3333, A 0.000, B 0.000, C 0.000 }
gfCNCPoint1[9261] = {X 121.4699, Y 14.7433, Z -1.3333, A 0.000, B 0.000, C 0.000 }
gfCNCPoint1[9262] = {X 120.9866, Y 15.5154, Z -1.3333, A 0.000, B 0.000, C 0.000 }
gfCNCPoint1[9263] = {X 120.3441, Y 16.1609, Z -1.3333, A 0.000, B 0.000, C 0.000 }
gfCNCPoint1[9264] = {X 120.3428, Y 41.0282, Z -1.3333, A 0.000, B 0.000, C 0.000 }
gfCNCPoint1[9265] = {X 120.4674, Y 41.1288, Z -1.3333, A 0.000, B 0.000, C 0.000 }
gfCNCPoint1[9266] = {X 121.0551, Y 41.7602, Z -1.3333, A 0.000, B 0.000, C 0.000 }
gfCNCPoint1[9267] = {X 121.4970, Y 42.5011, Z -1.3333, A 0.000, B 0.000, C 0.000 }
gfCNCPoint1[9268] = {X 121.7732, Y 43.3183, Z -1.3333, A 0.000, B 0.000, C 0.000 }
gfCNCPoint1[9269] = {X 121.8714, Y 44.1754, Z -1.3333, A 0.000, B 0.000, C 0.000 }
gfCNCPoint1[9270] = {X 121.8716, Y 45.0000, Z -1.3333, A 0.000, B 0.000, C 0.000 }
gfCNCPoint1[9271] = {X 121.7693, Y 45.9079, Z -1.3333, A 0.000, B 0.000, C 0.000 }
gfCNCPoint1[9272] = {X 121.4675, Y 46.7702, Z -1.3333, A 0.000, B 0.000, C 0.000 }
gfCNCPoint1[9273] = {X 120.9814, Y 47.5438, Z -1.3333, A 0.000, B 0.000, C 0.000 }
gfCNCPoint1[9274] = {X 120.3354, Y 48.1899, Z -1.3333, A 0.000, B 0.000, C 0.000 }
gfCNCPoint1[9275] = {X 119.5618, Y 48.6760, Z -1.3333, A 0.000, B 0.000, C 0.000 }
gfCNCPoint1[9276] = {X 118.6995, Y 48.9777, Z -1.3333, A 0.000, B 0.000, C 0.000 }
gfCNCPoint1[9277] = {X 117.7916, Y 49.0800, Z -1.3333, A 0.000, B 0.000, C 0.000 }
gfCNCPoint1[9278] = {X 111.9185, Y 49.0800, Z -1.3333, A 0.000, B 0.000, C 0.000 }
gfCNCPoint1[9279] = {X 111.0151, Y 48.9787, Z -1.3333, A 0.000, B 0.000, C 0.000 }
gfCNCPoint1[9280] = {X 110.1565, Y 48.6799, Z -1.3333, A 0.000, B 0.000, C 0.000 }
gfCNCPoint1[9281] = {X 109.3855, Y 48.1985, Z -1.3333, A 0.000, B 0.000, C 0.000 }
gfCNCPoint1[9282] = {X 108.7401, Y 47.5582, Z -1.3333, A 0.000, B 0.000, C 0.000 }
gfCNCPoint1[9283] = {X 108.2526, Y 46.7909, Z -1.3333, A 0.000, B 0.000, C 0.000 }
gfCNCPoint1[9284] = {X 107.9470, Y 45.9348, Z -1.3333, A 0.000, B 0.000, C 0.000 }
gfCNCPoint1[9285] = {X 107.8386, Y 45.0322, Z -1.3333, A 0.000, B 0.000, C 0.000 }
gfCNCPoint1[9286] = {X 107.8385, Y 44.1795, Z -1.3333, A 0.000, B 0.000, C 0.000 }
gfCNCPoint1[9287] = {X 107.8723, Y 43.6666, Z -1.3333, A 0.000, B 0.000, C 0.000 }
gfCNCPoint1[9288] = {X 107.9732, Y 43.1625, Z -1.3333, A 0.000, B 0.000, C 0.000 }
gfCNCPoint1[9289] = {X 108.1295, Y 42.6997, Z -1.3333, A 0.000, B 0.000, C 0.000 }
gfCNCPoint1[9290] = {X 108.3425, Y 42.2601, Z -1.3333, A 0.000, B 0.000, C 0.000 }
gfCNCPoint1[9291] = {X 108.8066, Y 41.5743, Z -1.3333, A 0.000, B 0.000, C 0.000 }
gfCNCPoint1[9292] = {X 109.3673, Y 40.9650, Z -1.3333, A 0.000, B 0.000, C 0.000 }
gfCNCPoint1[9293] = {X 109.3671, Y 39.0029, Z -1.3333, A 0.000, B 0.000, C 0.000 }
gfCNCPoint1[9294] = {X 108.9865, Y 39.0029, Z -1.3333, A 0.000, B 0.000, C 0.000 }
gfCNCPoint1[9295] = {X 105.8902, Y 46.5692, Z -1.3333, A 0.000, B 0.000, C 0.000 }
gfCNCPoint1[9296] = {X 105.5407, Y 47.2300, Z -1.3333, A 0.000, B 0.000, C 0.000 }
gfCNCPoint1[9297] = {X 105.0765, Y 47.8159, Z -1.3333, A 0.000, B 0.000, C 0.000 }
gfCNCPoint1[9298] = {X 104.5133, Y 48.3073, Z -1.3333, A 0.000, B 0.000, C 0.000 }
gfCNCPoint1[9299] = {X 103.8698, Y 48.6877, Z -1.3333, A 0.000, B 0.000, C 0.000 }
gfCNCPoint1[9300] = {X 102.9784, Y 48.9895, Z -1.3333, A 0.000, B 0.000, C 0.000 }
gfCNCPoint1[9301] = {X 102.0417, Y 49.0792, Z -1.3333, A 0.000, B 0.000, C 0.000 }
gfCNCPoint1[9302] = {X 101.1093, Y 48.9518, Z -1.3333, A 0.000, B 0.000, C 0.000 }
gfCNCPoint1[9303] = {X 100.2309, Y 48.6142, Z -1.3333, A 0.000, B 0.000, C 0.000 }
gfCNCPoint1[9304] = {X 99.4532, Y 48.0843, Z -1.3333, A 0.000, B 0.000, C 0.000 }
gfCNCPoint1[9305] = {X 98.8176, Y 47.3903, Z -1.3333, A 0.000, B 0.000, C 0.000 }
gfCNCPoint1[9306] = {X 98.3579, Y 46.5692, Z -1.3333, A 0.000, B 0.000, C 0.000 }
gfCNCPoint1[9307] = {X 94.8910, Y 38.0905, Z -1.3333, A 0.000, B 0.000, C 0.000 }
gfCNCPoint1[9308] = {X 94.8896, Y 38.2310, Z -1.3333, A 0.000, B 0.000, C 0.000 }
gfCNCPoint1[9309] = {X 94.8899, Y 41.0174, Z -1.3333, A 0.000, B 0.000, C 0.000 }
gfCNCPoint1[9310] = {X 95.4401, Y 41.5602, Z -1.3333, A 0.000, B 0.000, C 0.000 }
gfCNCPoint1[9311] = {X 95.8806, Y 42.1952, Z -1.3333, A 0.000, B 0.000, C 0.000 }
gfCNCPoint1[9312] = {X 96.1086, Y 42.6660, Z -1.3333, A 0.000, B 0.000, C 0.000 }
gfCNCPoint1[9313] = {X 96.2758, Y 43.1617, Z -1.3333, A 0.000, B 0.000, C 0.000 }
gfCNCPoint1[9314] = {X 96.3804, Y 43.6804, Z -1.3333, A 0.000, B 0.000, C 0.000 }
gfCNCPoint1[9315] = {X 96.4185, Y 44.2082, Z -1.3333, A 0.000, B 0.000, C 0.000 }
gfCNCPoint1[9316] = {X 96.4184, Y 45.0392, Z -1.3333, A 0.000, B 0.000, C 0.000 }
gfCNCPoint1[9317] = {X 96.3086, Y 45.9406, Z -1.3333, A 0.000, B 0.000, C 0.000 }
gfCNCPoint1[9318] = {X 96.0023, Y 46.7954, Z -1.3333, A 0.000, B 0.000, C 0.000 }
gfCNCPoint1[9319] = {X 95.5144, Y 47.5613, Z -1.3333, A 0.000, B 0.000, C 0.000 }
gfCNCPoint1[9320] = {X 94.8692, Y 48.2003, Z -1.3333, A 0.000, B 0.000, C 0.000 }
gfCNCPoint1[9321] = {X 94.0987, Y 48.6808, Z -1.3333, A 0.000, B 0.000, C 0.000 }
gfCNCPoint1[9322] = {X 93.2410, Y 48.9789, Z -1.3333, A 0.000, B 0.000, C 0.000 }
gfCNCPoint1[9323] = {X 92.3385, Y 49.0800, Z -1.3333, A 0.000, B 0.000, C 0.000 }
gfCNCPoint1[9324] = {X 85.8951, Y 49.0800, Z -1.3333, A 0.000, B 0.000, C 0.000 }
gfCNCPoint1[9325] = {X 84.9918, Y 48.9788, Z -1.3333, A 0.000, B 0.000, C 0.000 }
gfCNCPoint1[9326] = {X 84.1334, Y 48.6801, Z -1.3333, A 0.000, B 0.000, C 0.000 }
gfCNCPoint1[9327] = {X 83.3624, Y 48.1987, Z -1.3333, A 0.000, B 0.000, C 0.000 }
gfCNCPoint1[9328] = {X 82.7171, Y 47.5586, Z -1.3333, A 0.000, B 0.000, C 0.000 }
gfCNCPoint1[9329] = {X 82.2295, Y 46.7916, Z -1.3333, A 0.000, B 0.000, C 0.000 }
gfCNCPoint1[9330] = {X 81.9238, Y 45.9356, Z -1.3333, A 0.000, B 0.000, C 0.000 }
gfCNCPoint1[9331] = {X 81.8152, Y 45.0332, Z -1.3333, A 0.000, B 0.000, C 0.000 }
gfCNCPoint1[9332] = {X 81.8151, Y 44.2084, Z -1.3333, A 0.000, B 0.000, C 0.000 }
gfCNCPoint1[9333] = {X 81.9213, Y 43.3036, Z -1.3333, A 0.000, B 0.000, C 0.000 }
gfCNCPoint1[9334] = {X 82.2228, Y 42.4439, Z -1.3333, A 0.000, B 0.000, C 0.000 }
gfCNCPoint1[9335] = {X 82.7047, Y 41.6709, Z -1.3333, A 0.000, B 0.000, C 0.000 }
gfCNCPoint1[9336] = {X 83.3440, Y 41.0218, Z -1.3333, A 0.000, B 0.000, C 0.000 }
gfCNCPoint1[9337] = {X 83.3439, Y 28.5924, Z -1.3333, A 0.000, B 0.000, C 0.000 }
gfCNCPoint1[9338] = {X 79.3439, Y 28.5924, Z -1.3333, A 0.000, B 0.000, C 0.000 }
gfCNCPoint1[9339] = {X 83.4239, Y 28.5924, Z -1.3333, A 0.000, B 0.000, C 0.000 }
gfCNCPoint1[9340] = {X 83.4237, Y 16.1232, Z -1.3333, A 0.000, B 0.000, C 0.000 }
gfCNCPoint1[9341] = {X 82.7813, Y 15.4888, Z -1.3333, A 0.000, B 0.000, C 0.000 }
gfCNCPoint1[9342] = {X 82.2975, Y 14.7265, Z -1.3333, A 0.000, B 0.000, C 0.000 }
gfCNCPoint1[9343] = {X 81.9970, Y 13.8751, Z -1.3333, A 0.000, B 0.000, C 0.000 }
gfCNCPoint1[9344] = {X 81.8951, Y 12.9779, Z -1.3333, A 0.000, B 0.000, C 0.000 }
gfCNCPoint1[9345] = {X 81.8951, Y 12.1868, Z -1.3333, A 0.000, B 0.000, C 0.000 }
gfCNCPoint1[9346] = {X 81.9954, Y 11.2967, Z -1.3333, A 0.000, B 0.000, C 0.000 }
gfCNCPoint1[9347] = {X 82.2912, Y 10.4513, Z -1.3333, A 0.000, B 0.000, C 0.000 }
gfCNCPoint1[9348] = {X 82.7677, Y 9.6929, Z -1.3333, A 0.000, B 0.000, C 0.000 }
gfCNCPoint1[9349] = {X 83.4011, Y 9.0595, Z -1.3333, A 0.000, B 0.000, C 0.000 }
gfCNCPoint1[9350] = {X 84.1595, Y 8.5829, Z -1.3333, A 0.000, B 0.000, C 0.000 }
gfCNCPoint1[9351] = {X 85.0050, Y 8.2871, Z -1.3333, A 0.000, B 0.000, C 0.000 }
gfCNCPoint1[9352] = {X 85.8951, Y 8.1868, Z -1.3333, A 0.000, B 0.000, C 0.000 }
gfCNCPoint1[9353] = {X 94.0497, Y 8.1868, Z -1.3333, A 0.000, B 0.000, C 0.000 }
gfCNCPoint1[9354] = {X 94.9398, Y 8.2871, Z -1.3333, A 0.000, B 0.000, C 0.000 }
gfCNCPoint1[9355] = {X 95.7852, Y 8.5829, Z -1.3333, A 0.000, B 0.000, C 0.000 }
gfCNCPoint1[9356] = {X 96.5436, Y 9.0595, Z -1.3333, A 0.000, B 0.000, C 0.000 }
gfCNCPoint1[9357] = {X 97.1770, Y 9.6929, Z -1.3333, A 0.000, B 0.000, C 0.000 }
gfCNCPoint1[9358] = {X 97.6535, Y 10.4513, Z -1.3333, A 0.000, B 0.000, C 0.000 }
gfCNCPoint1[9359] = {X 97.9494, Y 11.2967, Z -1.3333, A 0.000, B 0.000, C 0.000 }
gfCNCPoint1[9360] = {X 98.0497, Y 12.1868, Z -1.3333, A 0.000, B 0.000, C 0.000 }
gfCNCPoint1[9361] = {X 98.0495, Y 13.0192, Z -1.3333, A 0.000, B 0.000, C 0.000 }
gfCNCPoint1[9362] = {X 97.9793, Y 13.7249, Z -1.3333, A 0.000, B 0.000, C 0.000 }
gfCNCPoint1[9363] = {X 97.7856, Y 14.4072, Z -1.3333, A 0.000, B 0.000, C 0.000 }
gfCNCPoint1[9364] = {X 97.4745, Y 15.0445, Z -1.3333, A 0.000, B 0.000, C 0.000 }
gfCNCPoint1[9365] = {X 97.4125, Y 15.1440, Z -1.3333, A 0.000, B 0.000, C 0.000 }
gfCNCPoint1[9366] = {X 97.3476, Y 15.2415, Z -1.3333, A 0.000, B 0.000, C 0.000 }
gfCNCPoint1[9367] = {X 97.4098, Y 15.3107, Z -1.3333, A 0.000, B 0.000, C 0.000 }
gfCNCPoint1[9368] = {X 97.9955, Y 16.7687, Z -1.3333, A 0.000, B 0.000, C 0.000 }
gfCNCPoint1[9369] = {X 101.3463, Y 25.0766, Z -1.3333, A 0.000, B 0.000, C 0.000 }
gfCNCPoint1[9370] = {X 101.8768, Y 26.3808, Z -1.3333, A 0.000, B 0.000, C 0.000 }
gfCNCPoint1[9371] = {X 102.1275, Y 25.7689, Z -1.3333, A 0.000, B 0.000, C 0.000 }
gfCNCPoint1[9372] = {X 106.3432, Y 15.2552, Z -1.3333, A 0.000, B 0.000, C 0.000 }
gfCNCPoint1[9373] = {X 106.3813, Y 15.1986, Z -1.3333, A 0.000, B 0.000, C 0.000 }
gfCNCPoint1[9374] = {X 106.3238, Y 15.1100, Z -1.3333, A 0.000, B 0.000, C 0.000 }
gfCNCPoint1[9375] = {X 106.2687, Y 15.0199, Z -1.3333, A 0.000, B 0.000, C 0.000 }
gfCNCPoint1[9376] = {X 105.9607, Y 14.3765, Z -1.3333, A 0.000, B 0.000, C 0.000 }
gfCNCPoint1[9377] = {X 105.7719, Y 13.6885, Z -1.3333, A 0.000, B 0.000, C 0.000 }
gfCNCPoint1[9378] = {X 105.7083, Y 12.9779, Z -1.3333, A 0.000, B 0.000, C 0.000 }
gfCNCPoint1[9379] = {X 105.7083, Y 12.1868, Z -1.3333, A 0.000, B 0.000, C 0.000 }
gfCNCPoint1[9380] = {X 105.8086, Y 11.2967, Z -1.3333, A 0.000, B 0.000, C 0.000 }
gfCNCPoint1[9381] = {X 106.1044, Y 10.4513, Z -1.3333, A 0.000, B 0.000, C 0.000 }
gfCNCPoint1[9382] = {X 106.5810, Y 9.6929, Z -1.3333, A 0.000, B 0.000, C 0.000 }
gfCNCPoint1[9383] = {X 107.2143, Y 9.0595, Z -1.3333, A 0.000, B 0.000, C 0.000 }
gfCNCPoint1[9384] = {X 107.9727, Y 8.5829, Z -1.3333, A 0.000, B 0.000, C 0.000 }
gfCNCPoint1[9385] = {X 108.8182, Y 8.2871, Z -1.3333, A 0.000, B 0.000, C 0.000 }
gfCNCPoint1[9386] = {X 109.7083, Y 8.1868, Z -1.3333, A 0.000, B 0.000, C 0.000 }
gfCNCPoint1[9387] = {X 117.7916, Y 8.1868, Z -1.3333, A 0.000, B 0.000, C 0.000 }
gfCNCPoint1[9388] = {X 118.6817, Y 8.2871, Z -1.3333, A 0.000, B 0.000, C 0.000 }
gfCNCPoint1[9389] = {X 119.5271, Y 8.5829, Z -1.3333, A 0.000, B 0.000, C 0.000 }
gfCNCPoint1[9390] = {X 120.2855, Y 9.0595, Z -1.3333, A 0.000, B 0.000, C 0.000 }
gfCNCPoint1[9391] = {X 120.9189, Y 9.6929, Z -1.3333, A 0.000, B 0.000, C 0.000 }
gfCNCPoint1[9392] = {X 121.3955, Y 10.4513, Z -1.3333, A 0.000, B 0.000, C 0.000 }
gfCNCPoint1[9393] = {X 121.6913, Y 11.2967, Z -1.3333, A 0.000, B 0.000, C 0.000 }
gfCNCPoint1[9394] = {X 121.7916, Y 12.1868, Z -1.3333, A 0.000, B 0.000, C 0.000 }
gfCNCPoint1[9395] = {X 121.7914, Y 13.0192, Z -1.3333, A 0.000, B 0.000, C 0.000 }
gfCNCPoint1[9396] = {X 121.6827, Y 13.9048, Z -1.3333, A 0.000, B 0.000, C 0.000 }
gfCNCPoint1[9397] = {X 121.3805, Y 14.7444, Z -1.3333, A 0.000, B 0.000, C 0.000 }
gfCNCPoint1[9398] = {X 120.8996, Y 15.4960, Z -1.3333, A 0.000, B 0.000, C 0.000 }
gfCNCPoint1[9399] = {X 120.2641, Y 16.1223, Z -1.3333, A 0.000, B 0.000, C 0.000 }
gfCNCPoint1[9400] = {X 120.2628, Y 41.0664, Z -1.3333, A 0.000, B 0.000, C 0.000 }
gfCNCPoint1[9401] = {X 120.4160, Y 41.1901, Z -1.3333, A 0.000, B 0.000, C 0.000 }
gfCNCPoint1[9402] = {X 120.9967, Y 41.8157, Z -1.3333, A 0.000, B 0.000, C 0.000 }
gfCNCPoint1[9403] = {X 121.4315, Y 42.5502, Z -1.3333, A 0.000, B 0.000, C 0.000 }
gfCNCPoint1[9404] = {X 121.7005, Y 43.3602, Z -1.3333, A 0.000, B 0.000, C 0.000 }
gfCNCPoint1[9405] = {X 121.7916, Y 44.2089, Z -1.3333, A 0.000, B 0.000, C 0.000 }
gfCNCPoint1[9406] = {X 121.7916, Y 45.0000, Z -1.3333, A 0.000, B 0.000, C 0.000 }
gfCNCPoint1[9407] = {X 121.6913, Y 45.8901, Z -1.3333, A 0.000, B 0.000, C 0.000 }
gfCNCPoint1[9408] = {X 121.3955, Y 46.7355, Z -1.3333, A 0.000, B 0.000, C 0.000 }
gfCNCPoint1[9409] = {X 120.9189, Y 47.4940, Z -1.3333, A 0.000, B 0.000, C 0.000 }
gfCNCPoint1[9410] = {X 120.2855, Y 48.1273, Z -1.3333, A 0.000, B 0.000, C 0.000 }
gfCNCPoint1[9411] = {X 119.5271, Y 48.6039, Z -1.3333, A 0.000, B 0.000, C 0.000 }
gfCNCPoint1[9412] = {X 118.6817, Y 48.8997, Z -1.3333, A 0.000, B 0.000, C 0.000 }
gfCNCPoint1[9413] = {X 117.7916, Y 49.0000, Z -1.3333, A 0.000, B 0.000, C 0.000 }
gfCNCPoint1[9414] = {X 111.9185, Y 49.0000, Z -1.3333, A 0.000, B 0.000, C 0.000 }
gfCNCPoint1[9415] = {X 111.0284, Y 48.8997, Z -1.3333, A 0.000, B 0.000, C 0.000 }
gfCNCPoint1[9416] = {X 110.1829, Y 48.6039, Z -1.3333, A 0.000, B 0.000, C 0.000 }
gfCNCPoint1[9417] = {X 109.4245, Y 48.1273, Z -1.3333, A 0.000, B 0.000, C 0.000 }
gfCNCPoint1[9418] = {X 108.7911, Y 47.4939, Z -1.3333, A 0.000, B 0.000, C 0.000 }
gfCNCPoint1[9419] = {X 108.3146, Y 46.7355, Z -1.3333, A 0.000, B 0.000, C 0.000 }
gfCNCPoint1[9420] = {X 108.0188, Y 45.8900, Z -1.3333, A 0.000, B 0.000, C 0.000 }
gfCNCPoint1[9421] = {X 107.9185, Y 45.0000, Z -1.3333, A 0.000, B 0.000, C 0.000 }
gfCNCPoint1[9422] = {X 107.9185, Y 44.1795, Z -1.3333, A 0.000, B 0.000, C 0.000 }
gfCNCPoint1[9423] = {X 107.9516, Y 43.6771, Z -1.3333, A 0.000, B 0.000, C 0.000 }
gfCNCPoint1[9424] = {X 108.0504, Y 43.1833, Z -1.3333, A 0.000, B 0.000, C 0.000 }
gfCNCPoint1[9425] = {X 108.2036, Y 42.7300, Z -1.3333, A 0.000, B 0.000, C 0.000 }
gfCNCPoint1[9426] = {X 108.4121, Y 42.2994, Z -1.3333, A 0.000, B 0.000, C 0.000 }
gfCNCPoint1[9427] = {X 108.4351, Y 42.2592, Z -1.3333, A 0.000, B 0.000, C 0.000 }
gfCNCPoint1[9428] = {X 108.4585, Y 42.2194, Z -1.3333, A 0.000, B 0.000, C 0.000 }
gfCNCPoint1[9429] = {X 108.9090, Y 41.5741, Z -1.3333, A 0.000, B 0.000, C 0.000 }
gfCNCPoint1[9430] = {X 109.4473, Y 40.9999, Z -1.3333, A 0.000, B 0.000, C 0.000 }
gfCNCPoint1[9431] = {X 109.4471, Y 38.9229, Z -1.3333, A 0.000, B 0.000, C 0.000 }
gfCNCPoint1[9432] = {X 108.9328, Y 38.9229, Z -1.3333, A 0.000, B 0.000, C 0.000 }
gfCNCPoint1[9433] = {X 105.8164, Y 46.5384, Z -1.3333, A 0.000, B 0.000, C 0.000 }
gfCNCPoint1[9434] = {X 105.3339, Y 47.3869, Z -1.3333, A 0.000, B 0.000, C 0.000 }
gfCNCPoint1[9435] = {X 104.6602, Y 48.0932, Z -1.3333, A 0.000, B 0.000, C 0.000 }
gfCNCPoint1[9436] = {X 103.8355, Y 48.6154, Z -1.3333, A 0.000, B 0.000, C 0.000 }
gfCNCPoint1[9437] = {X 102.9580, Y 48.9121, Z -1.3333, A 0.000, B 0.000, C 0.000 }
gfCNCPoint1[9438] = {X 102.0357, Y 48.9990, Z -1.3333, A 0.000, B 0.000, C 0.000 }
gfCNCPoint1[9439] = {X 101.1182, Y 48.8715, Z -1.3333, A 0.000, B 0.000, C 0.000 }
gfCNCPoint1[9440] = {X 100.2546, Y 48.5362, Z -1.3333, A 0.000, B 0.000, C 0.000 }
gfCNCPoint1[9441] = {X 99.4912, Y 48.0114, Z -1.3333, A 0.000, B 0.000, C 0.000 }
gfCNCPoint1[9442] = {X 98.8691, Y 47.3250, Z -1.3333, A 0.000, B 0.000, C 0.000 }
gfCNCPoint1[9443] = {X 98.4216, Y 46.5139, Z -1.3333, A 0.000, B 0.000, C 0.000 }
gfCNCPoint1[9444] = {X 94.8147, Y 37.6927, Z -1.3333, A 0.000, B 0.000, C 0.000 }
gfCNCPoint1[9445] = {X 94.8096, Y 38.2306, Z -1.3333, A 0.000, B 0.000, C 0.000 }
gfCNCPoint1[9446] = {X 94.8099, Y 41.0556, Z -1.3333, A 0.000, B 0.000, C 0.000 }
gfCNCPoint1[9447] = {X 95.3667, Y 41.5973, Z -1.3333, A 0.000, B 0.000, C 0.000 }
gfCNCPoint1[9448] = {X 95.8109, Y 42.2345, Z -1.3333, A 0.000, B 0.000, C 0.000 }
gfCNCPoint1[9449] = {X 96.0345, Y 42.6963, Z -1.3333, A 0.000, B 0.000, C 0.000 }
gfCNCPoint1[9450] = {X 96.1985, Y 43.1824, Z -1.3333, A 0.000, B 0.000, C 0.000 }
gfCNCPoint1[9451] = {X 96.3012, Y 43.6912, Z -1.3333, A 0.000, B 0.000, C 0.000 }
gfCNCPoint1[9452] = {X 96.3385, Y 44.2089, Z -1.3333, A 0.000, B 0.000, C 0.000 }
gfCNCPoint1[9453] = {X 96.3384, Y 45.0384, Z -1.3333, A 0.000, B 0.000, C 0.000 }
gfCNCPoint1[9454] = {X 96.2308, Y 45.9222, Z -1.3333, A 0.000, B 0.000, C 0.000 }
gfCNCPoint1[9455] = {X 95.9304, Y 46.7602, Z -1.3333, A 0.000, B 0.000, C 0.000 }
gfCNCPoint1[9456] = {X 95.4521, Y 47.5111, Z -1.3333, A 0.000, B 0.000, C 0.000 }
gfCNCPoint1[9457] = {X 94.8196, Y 48.1376, Z -1.3333, A 0.000, B 0.000, C 0.000 }
gfCNCPoint1[9458] = {X 94.0642, Y 48.6086, Z -1.3333, A 0.000, B 0.000, C 0.000 }
gfCNCPoint1[9459] = {X 93.2233, Y 48.9009, Z -1.3333, A 0.000, B 0.000, C 0.000 }
gfCNCPoint1[9460] = {X 92.3385, Y 49.0000, Z -1.3333, A 0.000, B 0.000, C 0.000 }
gfCNCPoint1[9461] = {X 85.8951, Y 49.0000, Z -1.3333, A 0.000, B 0.000, C 0.000 }
gfCNCPoint1[9462] = {X 85.0050, Y 48.8997, Z -1.3333, A 0.000, B 0.000, C 0.000 }
gfCNCPoint1[9463] = {X 84.1595, Y 48.6039, Z -1.3333, A 0.000, B 0.000, C 0.000 }
gfCNCPoint1[9464] = {X 83.4011, Y 48.1273, Z -1.3333, A 0.000, B 0.000, C 0.000 }
gfCNCPoint1[9465] = {X 82.7677, Y 47.4939, Z -1.3333, A 0.000, B 0.000, C 0.000 }
gfCNCPoint1[9466] = {X 82.2912, Y 46.7355, Z -1.3333, A 0.000, B 0.000, C 0.000 }
gfCNCPoint1[9467] = {X 81.9954, Y 45.8900, Z -1.3333, A 0.000, B 0.000, C 0.000 }
gfCNCPoint1[9468] = {X 81.8951, Y 45.0000, Z -1.3333, A 0.000, B 0.000, C 0.000 }
gfCNCPoint1[9469] = {X 81.8951, Y 44.2089, Z -1.3333, A 0.000, B 0.000, C 0.000 }
gfCNCPoint1[9470] = {X 82.0014, Y 43.3124, Z -1.3333, A 0.000, B 0.000, C 0.000 }
gfCNCPoint1[9471] = {X 82.3031, Y 42.4615, Z -1.3333, A 0.000, B 0.000, C 0.000 }
gfCNCPoint1[9472] = {X 82.7852, Y 41.6981, Z -1.3333, A 0.000, B 0.000, C 0.000 }
gfCNCPoint1[9473] = {X 83.4240, Y 41.0601, Z -1.3333, A 0.000, B 0.000, C 0.000 }
gfCNCPoint1[9474] = {X 83.4239, Y 28.5924, Z -1.3333, A 0.000, B 0.000, C 0.000 }
gfCNCPoint1[9475] = {X 79.3439, Y 28.5924, Z -1.3333, A 0.000, B 0.000, C 0.000 }
gfCNCPoint1[9476] = {X 79.3439, Y 28.5924, Z 1.6667, A 0.000, B 0.000, C 0.000 }
gfCNCPoint1[9477] = {X 79.3439, Y 28.5924, Z 11.0000, A 0.000, B 0.000, C 0.000 }
gfCNCPoint1[9478] = {X 136.1636, Y 30.3961, Z 11.0000, A 0.000, B 0.000, C 0.000 }
gfCNCPoint1[9479] = {X 136.1636, Y 30.3961, Z 1.6667, A 0.000, B 0.000, C 0.000 }
gfCNCPoint1[9480] = {X 136.1636, Y 30.3961, Z -1.3333, A 0.000, B 0.000, C 0.000 }
gfCNCPoint1[9481] = {X 140.2436, Y 30.3961, Z -1.3333, A 0.000, B 0.000, C 0.000 }
gfCNCPoint1[9482] = {X 140.2436, Y 19.8765, Z -1.3333, A 0.000, B 0.000, C 0.000 }
gfCNCPoint1[9483] = {X 137.4245, Y 19.8762, Z -1.3333, A 0.000, B 0.000, C 0.000 }
gfCNCPoint1[9484] = {X 136.8921, Y 20.5211, Z -1.3333, A 0.000, B 0.000, C 0.000 }
gfCNCPoint1[9485] = {X 136.2454, Y 21.0514, Z -1.3333, A 0.000, B 0.000, C 0.000 }
gfCNCPoint1[9486] = {X 135.5087, Y 21.4472, Z -1.3333, A 0.000, B 0.000, C 0.000 }
gfCNCPoint1[9487] = {X 134.7095, Y 21.6936, Z -1.3333, A 0.000, B 0.000, C 0.000 }
gfCNCPoint1[9488] = {X 133.8778, Y 21.7814, Z -1.3333, A 0.000, B 0.000, C 0.000 }
gfCNCPoint1[9489] = {X 133.2006, Y 21.7815, Z -1.3333, A 0.000, B 0.000, C 0.000 }
gfCNCPoint1[9490] = {X 132.2394, Y 21.6732, Z -1.3333, A 0.000, B 0.000, C 0.000 }
gfCNCPoint1[9491] = {X 131.3263, Y 21.3537, Z -1.3333, A 0.000, B 0.000, C 0.000 }
gfCNCPoint1[9492] = {X 130.5072, Y 20.8390, Z -1.3333, A 0.000, B 0.000, C 0.000 }
gfCNCPoint1[9493] = {X 129.8231, Y 20.1550, Z -1.3333, A 0.000, B 0.000, C 0.000 }
gfCNCPoint1[9494] = {X 129.3085, Y 19.3359, Z -1.3333, A 0.000, B 0.000, C 0.000 }
gfCNCPoint1[9495] = {X 128.9890, Y 18.4228, Z -1.3333, A 0.000, B 0.000, C 0.000 }
gfCNCPoint1[9496] = {X 128.8806, Y 17.4615, Z -1.3333, A 0.000, B 0.000, C 0.000 }
gfCNCPoint1[9497] = {X 128.8806, Y 10.4835, Z -1.3333, A 0.000, B 0.000, C 0.000 }
gfCNCPoint1[9498] = {X 128.9874, Y 9.5289, Z -1.3333, A 0.000, B 0.000, C 0.000 }
gfCNCPoint1[9499] = {X 129.3026, Y 8.6214, Z -1.3333, A 0.000, B 0.000, C 0.000 }
gfCNCPoint1[9500] = {X 129.8104, Y 7.8061, Z -1.3333, A 0.000, B 0.000, C 0.000 }
gfCNCPoint1[9501] = {X 130.4859, Y 7.1231, Z -1.3333, A 0.000, B 0.000, C 0.000 }
gfCNCPoint1[9502] = {X 131.2956, Y 6.6063, Z -1.3333, A 0.000, B 0.000, C 0.000 }
gfCNCPoint1[9503] = {X 132.1995, Y 6.2811, Z -1.3333, A 0.000, B 0.000, C 0.000 }
gfCNCPoint1[9504] = {X 133.1529, Y 6.1638, Z -1.3333, A 0.000, B 0.000, C 0.000 }
gfCNCPoint1[9505] = {X 133.8866, Y 6.1637, Z -1.3333, A 0.000, B 0.000, C 0.000 }
gfCNCPoint1[9506] = {X 134.7114, Y 6.2518, Z -1.3333, A 0.000, B 0.000, C 0.000 }
gfCNCPoint1[9507] = {X 135.5041, Y 6.4959, Z -1.3333, A 0.000, B 0.000, C 0.000 }
gfCNCPoint1[9508] = {X 136.2356, Y 6.8870, Z -1.3333, A 0.000, B 0.000, C 0.000 }
gfCNCPoint1[9509] = {X 136.8788, Y 7.4107, Z -1.3333, A 0.000, B 0.000, C 0.000 }
gfCNCPoint1[9510] = {X 137.4101, Y 8.0477, Z -1.3333, A 0.000, B 0.000, C 0.000 }
gfCNCPoint1[9511] = {X 155.1119, Y 8.0488, Z -1.3333, A 0.000, B 0.000, C 0.000 }
gfCNCPoint1[9512] = {X 155.6439, Y 7.4107, Z -1.3333, A 0.000, B 0.000, C 0.000 }
gfCNCPoint1[9513] = {X 156.2882, Y 6.8863, Z -1.3333, A 0.000, B 0.000, C 0.000 }
gfCNCPoint1[9514] = {X 157.0210, Y 6.4950, Z -1.3333, A 0.000, B 0.000, C 0.000 }
gfCNCPoint1[9515] = {X 157.8151, Y 6.2511, Z -1.3333, A 0.000, B 0.000, C 0.000 }
gfCNCPoint1[9516] = {X 158.6412, Y 6.1637, Z -1.3333, A 0.000, B 0.000, C 0.000 }
gfCNCPoint1[9517] = {X 159.3781, Y 6.1639, Z -1.3333, A 0.000, B 0.000, C 0.000 }
gfCNCPoint1[9518] = {X 160.3301, Y 6.2828, Z -1.3333, A 0.000, B 0.000, C 0.000 }
gfCNCPoint1[9519] = {X 161.2324, Y 6.6088, Z -1.3333, A 0.000, B 0.000, C 0.000 }
gfCNCPoint1[9520] = {X 162.0405, Y 7.1260, Z -1.3333, A 0.000, B 0.000, C 0.000 }
gfCNCPoint1[9521] = {X 162.7145, Y 7.8088, Z -1.3333, A 0.000, B 0.000, C 0.000 }
gfCNCPoint1[9522] = {X 163.2212, Y 8.6236, Z -1.3333, A 0.000, B 0.000, C 0.000 }
gfCNCPoint1[9523] = {X 163.5355, Y 9.5300, Z -1.3333, A 0.000, B 0.000, C 0.000 }
gfCNCPoint1[9524] = {X 163.6421, Y 10.4835, Z -1.3333, A 0.000, B 0.000, C 0.000 }
gfCNCPoint1[9525] = {X 163.6421, Y 17.4615, Z -1.3333, A 0.000, B 0.000, C 0.000 }
gfCNCPoint1[9526] = {X 163.5355, Y 18.4152, Z -1.3333, A 0.000, B 0.000, C 0.000 }
gfCNCPoint1[9527] = {X 163.2211, Y 19.3218, Z -1.3333, A 0.000, B 0.000, C 0.000 }
gfCNCPoint1[9528] = {X 162.7142, Y 20.1366, Z -1.3333, A 0.000, B 0.000, C 0.000 }
gfCNCPoint1[9529] = {X 162.0400, Y 20.8194, Z -1.3333, A 0.000, B 0.000, C 0.000 }
gfCNCPoint1[9530] = {X 161.2318, Y 21.3365, Z -1.3333, A 0.000, B 0.000, C 0.000 }
gfCNCPoint1[9531] = {X 160.3292, Y 21.6625, Z -1.3333, A 0.000, B 0.000, C 0.000 }
gfCNCPoint1[9532] = {X 159.3770, Y 21.7812, Z -1.3333, A 0.000, B 0.000, C 0.000 }
gfCNCPoint1[9533] = {X 158.6789, Y 21.7815, Z -1.3333, A 0.000, B 0.000, C 0.000 }
gfCNCPoint1[9534] = {X 157.8407, Y 21.6958, Z -1.3333, A 0.000, B 0.000, C 0.000 }
gfCNCPoint1[9535] = {X 157.0346, Y 21.4504, Z -1.3333, A 0.000, B 0.000, C 0.000 }
gfCNCPoint1[9536] = {X 156.2907, Y 21.0545, Z -1.3333, A 0.000, B 0.000, C 0.000 }
gfCNCPoint1[9537] = {X 155.6369, Y 20.5230, Z -1.3333, A 0.000, B 0.000, C 0.000 }
gfCNCPoint1[9538] = {X 155.0975, Y 19.8756, Z -1.3333, A 0.000, B 0.000, C 0.000 }
gfCNCPoint1[9539] = {X 152.2755, Y 19.8771, Z -1.3333, A 0.000, B 0.000, C 0.000 }
gfCNCPoint1[9540] = {X 152.2738, Y 40.8742, Z -1.3333, A 0.000, B 0.000, C 0.000 }
gfCNCPoint1[9541] = {X 152.7410, Y 41.3771, Z -1.3333, A 0.000, B 0.000, C 0.000 }
gfCNCPoint1[9542] = {X 152.8347, Y 41.4890, Z -1.3333, A 0.000, B 0.000, C 0.000 }
gfCNCPoint1[9543] = {X 153.3600, Y 42.3143, Z -1.3333, A 0.000, B 0.000, C 0.000 }
gfCNCPoint1[9544] = {X 153.6883, Y 43.2357, Z -1.3333, A 0.000, B 0.000, C 0.000 }
gfCNCPoint1[9545] = {X 153.8031, Y 44.2072, Z -1.3333, A 0.000, B 0.000, C 0.000 }
gfCNCPoint1[9546] = {X 153.8029, Y 45.0415, Z -1.3333, A 0.000, B 0.000, C 0.000 }
gfCNCPoint1[9547] = {X 153.6867, Y 45.9960, Z -1.3333, A 0.000, B 0.000, C 0.000 }
gfCNCPoint1[9548] = {X 153.3623, Y 46.9011, Z -1.3333, A 0.000, B 0.000, C 0.000 }
gfCNCPoint1[9549] = {X 152.8458, Y 47.7120, Z -1.3333, A 0.000, B 0.000, C 0.000 }
gfCNCPoint1[9550] = {X 152.1626, Y 48.3886, Z -1.3333, A 0.000, B 0.000, C 0.000 }
gfCNCPoint1[9551] = {X 151.3468, Y 48.8973, Z -1.3333, A 0.000, B 0.000, C 0.000 }
gfCNCPoint1[9552] = {X 150.4386, Y 49.2130, Z -1.3333, A 0.000, B 0.000, C 0.000 }
gfCNCPoint1[9553] = {X 149.4831, Y 49.3200, Z -1.3333, A 0.000, B 0.000, C 0.000 }
gfCNCPoint1[9554] = {X 143.0396, Y 49.3200, Z -1.3333, A 0.000, B 0.000, C 0.000 }
gfCNCPoint1[9555] = {X 142.0831, Y 49.2128, Z -1.3333, A 0.000, B 0.000, C 0.000 }
gfCNCPoint1[9556] = {X 141.1741, Y 48.8964, Z -1.3333, A 0.000, B 0.000, C 0.000 }
gfCNCPoint1[9557] = {X 140.3576, Y 48.3866, Z -1.3333, A 0.000, B 0.000, C 0.000 }
gfCNCPoint1[9558] = {X 139.6743, Y 47.7087, Z -1.3333, A 0.000, B 0.000, C 0.000 }
gfCNCPoint1[9559] = {X 139.1581, Y 46.8964, Z -1.3333, A 0.000, B 0.000, C 0.000 }
gfCNCPoint1[9560] = {X 138.8346, Y 45.9899, Z -1.3333, A 0.000, B 0.000, C 0.000 }
gfCNCPoint1[9561] = {X 138.7198, Y 45.0342, Z -1.3333, A 0.000, B 0.000, C 0.000 }
gfCNCPoint1[9562] = {X 138.7200, Y 44.1494, Z -1.3333, A 0.000, B 0.000, C 0.000 }
gfCNCPoint1[9563] = {X 138.8305, Y 43.2364, Z -1.3333, A 0.000, B 0.000, C 0.000 }
gfCNCPoint1[9564] = {X 139.1317, Y 42.3675, Z -1.3333, A 0.000, B 0.000, C 0.000 }
gfCNCPoint1[9565] = {X 139.6099, Y 41.5821, Z -1.3333, A 0.000, B 0.000, C 0.000 }
gfCNCPoint1[9566] = {X 140.2436, Y 40.9157, Z -1.3333, A 0.000, B 0.000, C 0.000 }
gfCNCPoint1[9567] = {X 140.2436, Y 30.3961, Z -1.3333, A 0.000, B 0.000, C 0.000 }
gfCNCPoint1[9568] = {X 136.2436, Y 30.3961, Z -1.3333, A 0.000, B 0.000, C 0.000 }
gfCNCPoint1[9569] = {X 140.3236, Y 30.3961, Z -1.3333, A 0.000, B 0.000, C 0.000 }
gfCNCPoint1[9570] = {X 140.3236, Y 19.7965, Z -1.3333, A 0.000, B 0.000, C 0.000 }
gfCNCPoint1[9571] = {X 137.3802, Y 19.7956, Z -1.3333, A 0.000, B 0.000, C 0.000 }
gfCNCPoint1[9572] = {X 137.3572, Y 19.8328, Z -1.3333, A 0.000, B 0.000, C 0.000 }
gfCNCPoint1[9573] = {X 136.8347, Y 20.4654, Z -1.3333, A 0.000, B 0.000, C 0.000 }
gfCNCPoint1[9574] = {X 136.2001, Y 20.9855, Z -1.3333, A 0.000, B 0.000, C 0.000 }
gfCNCPoint1[9575] = {X 135.4772, Y 21.3737, Z -1.3333, A 0.000, B 0.000, C 0.000 }
gfCNCPoint1[9576] = {X 134.6931, Y 21.6153, Z -1.3333, A 0.000, B 0.000, C 0.000 }
gfCNCPoint1[9577] = {X 133.8772, Y 21.7014, Z -1.3333, A 0.000, B 0.000, C 0.000 }
gfCNCPoint1[9578] = {X 133.2006, Y 21.7015, Z -1.3333, A 0.000, B 0.000, C 0.000 }
gfCNCPoint1[9579] = {X 132.2572, Y 21.5952, Z -1.3333, A 0.000, B 0.000, C 0.000 }
gfCNCPoint1[9580] = {X 131.3610, Y 21.2816, Z -1.3333, A 0.000, B 0.000, C 0.000 }
gfCNCPoint1[9581] = {X 130.5570, Y 20.7765, Z -1.3333, A 0.000, B 0.000, C 0.000 }
gfCNCPoint1[9582] = {X 129.8857, Y 20.1051, Z -1.3333, A 0.000, B 0.000, C 0.000 }
gfCNCPoint1[9583] = {X 129.3805, Y 19.3012, Z -1.3333, A 0.000, B 0.000, C 0.000 }
gfCNCPoint1[9584] = {X 129.0669, Y 18.4050, Z -1.3333, A 0.000, B 0.000, C 0.000 }
gfCNCPoint1[9585] = {X 128.9606, Y 17.4615, Z -1.3333, A 0.000, B 0.000, C 0.000 }
gfCNCPoint1[9586] = {X 128.9606, Y 10.4835, Z -1.3333, A 0.000, B 0.000, C 0.000 }
gfCNCPoint1[9587] = {X 129.0655, Y 9.5466, Z -1.3333, A 0.000, B 0.000, C 0.000 }
gfCNCPoint1[9588] = {X 129.3747, Y 8.6559, Z -1.3333, A 0.000, B 0.000, C 0.000 }
gfCNCPoint1[9589] = {X 129.8732, Y 7.8557, Z -1.3333, A 0.000, B 0.000, C 0.000 }
gfCNCPoint1[9590] = {X 130.5362, Y 7.1853, Z -1.3333, A 0.000, B 0.000, C 0.000 }
gfCNCPoint1[9591] = {X 131.3309, Y 6.6781, Z -1.3333, A 0.000, B 0.000, C 0.000 }
gfCNCPoint1[9592] = {X 132.2180, Y 6.3589, Z -1.3333, A 0.000, B 0.000, C 0.000 }
gfCNCPoint1[9593] = {X 133.1538, Y 6.2438, Z -1.3333, A 0.000, B 0.000, C 0.000 }
gfCNCPoint1[9594] = {X 133.8858, Y 6.2437, Z -1.3333, A 0.000, B 0.000, C 0.000 }
gfCNCPoint1[9595] = {X 134.7035, Y 6.3319, Z -1.3333, A 0.000, B 0.000, C 0.000 }
gfCNCPoint1[9596] = {X 135.4889, Y 6.5763, Z -1.3333, A 0.000, B 0.000, C 0.000 }
gfCNCPoint1[9597] = {X 136.2122, Y 6.9677, Z -1.3333, A 0.000, B 0.000, C 0.000 }
gfCNCPoint1[9598] = {X 136.8464, Y 7.4914, Z -1.3333, A 0.000, B 0.000, C 0.000 }
gfCNCPoint1[9599] = {X 137.3676, Y 8.1277, Z -1.3333, A 0.000, B 0.000, C 0.000 }
gfCNCPoint1[9600] = {X 155.1544, Y 8.1288, Z -1.3333, A 0.000, B 0.000, C 0.000 }
gfCNCPoint1[9601] = {X 155.6763, Y 7.4914, Z -1.3333, A 0.000, B 0.000, C 0.000 }
gfCNCPoint1[9602] = {X 156.3115, Y 6.9670, Z -1.3333, A 0.000, B 0.000, C 0.000 }
gfCNCPoint1[9603] = {X 157.0362, Y 6.5753, Z -1.3333, A 0.000, B 0.000, C 0.000 }
gfCNCPoint1[9604] = {X 157.8229, Y 6.3311, Z -1.3333, A 0.000, B 0.000, C 0.000 }
gfCNCPoint1[9605] = {X 158.6420, Y 6.2437, Z -1.3333, A 0.000, B 0.000, C 0.000 }
gfCNCPoint1[9606] = {X 159.3770, Y 6.2439, Z -1.3333, A 0.000, B 0.000, C 0.000 }
gfCNCPoint1[9607] = {X 160.3114, Y 6.3606, Z -1.3333, A 0.000, B 0.000, C 0.000 }
gfCNCPoint1[9608] = {X 161.1970, Y 6.6806, Z -1.3333, A 0.000, B 0.000, C 0.000 }
gfCNCPoint1[9609] = {X 161.9902, Y 7.1882, Z -1.3333, A 0.000, B 0.000, C 0.000 }
gfCNCPoint1[9610] = {X 162.6517, Y 7.8584, Z -1.3333, A 0.000, B 0.000, C 0.000 }
gfCNCPoint1[9611] = {X 163.1490, Y 8.6580, Z -1.3333, A 0.000, B 0.000, C 0.000 }
gfCNCPoint1[9612] = {X 163.4575, Y 9.5477, Z -1.3333, A 0.000, B 0.000, C 0.000 }
gfCNCPoint1[9613] = {X 163.5621, Y 10.4835, Z -1.3333, A 0.000, B 0.000, C 0.000 }
gfCNCPoint1[9614] = {X 163.5621, Y 17.4615, Z -1.3333, A 0.000, B 0.000, C 0.000 }
gfCNCPoint1[9615] = {X 163.4575, Y 18.3975, Z -1.3333, A 0.000, B 0.000, C 0.000 }
gfCNCPoint1[9616] = {X 163.1489, Y 19.2873, Z -1.3333, A 0.000, B 0.000, C 0.000 }
gfCNCPoint1[9617] = {X 162.6514, Y 20.0870, Z -1.3333, A 0.000, B 0.000, C 0.000 }
gfCNCPoint1[9618] = {X 161.9897, Y 20.7572, Z -1.3333, A 0.000, B 0.000, C 0.000 }
gfCNCPoint1[9619] = {X 161.1964, Y 21.2648, Z -1.3333, A 0.000, B 0.000, C 0.000 }
gfCNCPoint1[9620] = {X 160.3106, Y 21.5847, Z -1.3333, A 0.000, B 0.000, C 0.000 }
gfCNCPoint1[9621] = {X 159.3760, Y 21.7012, Z -1.3333, A 0.000, B 0.000, C 0.000 }
gfCNCPoint1[9622] = {X 158.6793, Y 21.7015, Z -1.3333, A 0.000, B 0.000, C 0.000 }
gfCNCPoint1[9623] = {X 157.8482, Y 21.6157, Z -1.3333, A 0.000, B 0.000, C 0.000 }
gfCNCPoint1[9624] = {X 157.0496, Y 21.3700, Z -1.3333, A 0.000, B 0.000, C 0.000 }
gfCNCPoint1[9625] = {X 156.3139, Y 20.9738, Z -1.3333, A 0.000, B 0.000, C 0.000 }
gfCNCPoint1[9626] = {X 155.6692, Y 20.4423, Z -1.3333, A 0.000, B 0.000, C 0.000 }
gfCNCPoint1[9627] = {X 155.1400, Y 19.7956, Z -1.3333, A 0.000, B 0.000, C 0.000 }
gfCNCPoint1[9628] = {X 152.1955, Y 19.7972, Z -1.3333, A 0.000, B 0.000, C 0.000 }
gfCNCPoint1[9629] = {X 152.1938, Y 40.9056, Z -1.3333, A 0.000, B 0.000, C 0.000 }
gfCNCPoint1[9630] = {X 152.6810, Y 41.4300, Z -1.3333, A 0.000, B 0.000, C 0.000 }
gfCNCPoint1[9631] = {X 152.7729, Y 41.5398, Z -1.3333, A 0.000, B 0.000, C 0.000 }
gfCNCPoint1[9632] = {X 153.2883, Y 42.3498, Z -1.3333, A 0.000, B 0.000, C 0.000 }
gfCNCPoint1[9633] = {X 153.6104, Y 43.2542, Z -1.3333, A 0.000, B 0.000, C 0.000 }
gfCNCPoint1[9634] = {X 153.7231, Y 44.2076, Z -1.3333, A 0.000, B 0.000, C 0.000 }
gfCNCPoint1[9635] = {X 153.7229, Y 45.0408, Z -1.3333, A 0.000, B 0.000, C 0.000 }
gfCNCPoint1[9636] = {X 153.6089, Y 45.9775, Z -1.3333, A 0.000, B 0.000, C 0.000 }
gfCNCPoint1[9637] = {X 153.2905, Y 46.8659, Z -1.3333, A 0.000, B 0.000, C 0.000 }
gfCNCPoint1[9638] = {X 152.7835, Y 47.6618, Z -1.3333, A 0.000, B 0.000, C 0.000 }
gfCNCPoint1[9639] = {X 152.1130, Y 48.3258, Z -1.3333, A 0.000, B 0.000, C 0.000 }
gfCNCPoint1[9640] = {X 151.3123, Y 48.8251, Z -1.3333, A 0.000, B 0.000, C 0.000 }
gfCNCPoint1[9641] = {X 150.4209, Y 49.1350, Z -1.3333, A 0.000, B 0.000, C 0.000 }
gfCNCPoint1[9642] = {X 149.4831, Y 49.2400, Z -1.3333, A 0.000, B 0.000, C 0.000 }
gfCNCPoint1[9643] = {X 143.0396, Y 49.2400, Z -1.3333, A 0.000, B 0.000, C 0.000 }
gfCNCPoint1[9644] = {X 142.1008, Y 49.1348, Z -1.3333, A 0.000, B 0.000, C 0.000 }
gfCNCPoint1[9645] = {X 141.2086, Y 48.8243, Z -1.3333, A 0.000, B 0.000, C 0.000 }
gfCNCPoint1[9646] = {X 140.4073, Y 48.3239, Z -1.3333, A 0.000, B 0.000, C 0.000 }
gfCNCPoint1[9647] = {X 139.7367, Y 47.6586, Z -1.3333, A 0.000, B 0.000, C 0.000 }
gfCNCPoint1[9648] = {X 139.2300, Y 46.8612, Z -1.3333, A 0.000, B 0.000, C 0.000 }
gfCNCPoint1[9649] = {X 138.9124, Y 45.9715, Z -1.3333, A 0.000, B 0.000, C 0.000 }
gfCNCPoint1[9650] = {X 138.7998, Y 45.0336, Z -1.3333, A 0.000, B 0.000, C 0.000 }
gfCNCPoint1[9651] = {X 138.8000, Y 44.1505, Z -1.3333, A 0.000, B 0.000, C 0.000 }
gfCNCPoint1[9652] = {X 138.9105, Y 43.2454, Z -1.3333, A 0.000, B 0.000, C 0.000 }
gfCNCPoint1[9653] = {X 139.2119, Y 42.3850, Z -1.3333, A 0.000, B 0.000, C 0.000 }
gfCNCPoint1[9654] = {X 139.6903, Y 41.6088, Z -1.3333, A 0.000, B 0.000, C 0.000 }
gfCNCPoint1[9655] = {X 140.3236, Y 40.9529, Z -1.3333, A 0.000, B 0.000, C 0.000 }
gfCNCPoint1[9656] = {X 140.3236, Y 30.3961, Z -1.3333, A 0.000, B 0.000, C 0.000 }
gfCNCPoint1[9657] = {X 136.3236, Y 30.3961, Z -1.3333, A 0.000, B 0.000, C 0.000 }
gfCNCPoint1[9658] = {X 140.4036, Y 30.3961, Z -1.3333, A 0.000, B 0.000, C 0.000 }
gfCNCPoint1[9659] = {X 140.4036, Y 19.7166, Z -1.3333, A 0.000, B 0.000, C 0.000 }
gfCNCPoint1[9660] = {X 137.3355, Y 19.7156, Z -1.3333, A 0.000, B 0.000, C 0.000 }
gfCNCPoint1[9661] = {X 137.2900, Y 19.7895, Z -1.3333, A 0.000, B 0.000, C 0.000 }
gfCNCPoint1[9662] = {X 136.7773, Y 20.4097, Z -1.3333, A 0.000, B 0.000, C 0.000 }
gfCNCPoint1[9663] = {X 136.1548, Y 20.9196, Z -1.3333, A 0.000, B 0.000, C 0.000 }
gfCNCPoint1[9664] = {X 135.4458, Y 21.3001, Z -1.3333, A 0.000, B 0.000, C 0.000 }
gfCNCPoint1[9665] = {X 134.6767, Y 21.5370, Z -1.3333, A 0.000, B 0.000, C 0.000 }
gfCNCPoint1[9666] = {X 133.8765, Y 21.6214, Z -1.3333, A 0.000, B 0.000, C 0.000 }
gfCNCPoint1[9667] = {X 133.2006, Y 21.6215, Z -1.3333, A 0.000, B 0.000, C 0.000 }
gfCNCPoint1[9668] = {X 132.2750, Y 21.5172, Z -1.3333, A 0.000, B 0.000, C 0.000 }
gfCNCPoint1[9669] = {X 131.3957, Y 21.2096, Z -1.3333, A 0.000, B 0.000, C 0.000 }
gfCNCPoint1[9670] = {X 130.6069, Y 20.7140, Z -1.3333, A 0.000, B 0.000, C 0.000 }
gfCNCPoint1[9671] = {X 129.9482, Y 20.0553, Z -1.3333, A 0.000, B 0.000, C 0.000 }
gfCNCPoint1[9672] = {X 129.4526, Y 19.2665, Z -1.3333, A 0.000, B 0.000, C 0.000 }
gfCNCPoint1[9673] = {X 129.1449, Y 18.3872, Z -1.3333, A 0.000, B 0.000, C 0.000 }
gfCNCPoint1[9674] = {X 129.0406, Y 17.4615, Z -1.3333, A 0.000, B 0.000, C 0.000 }
gfCNCPoint1[9675] = {X 129.0406, Y 10.4835, Z -1.3333, A 0.000, B 0.000, C 0.000 }
gfCNCPoint1[9676] = {X 129.1435, Y 9.5642, Z -1.3333, A 0.000, B 0.000, C 0.000 }
gfCNCPoint1[9677] = {X 129.4469, Y 8.6904, Z -1.3333, A 0.000, B 0.000, C 0.000 }
gfCNCPoint1[9678] = {X 129.9360, Y 7.9052, Z -1.3333, A 0.000, B 0.000, C 0.000 }
gfCNCPoint1[9679] = {X 130.5864, Y 7.2475, Z -1.3333, A 0.000, B 0.000, C 0.000 }
gfCNCPoint1[9680] = {X 131.3662, Y 6.7499, Z -1.3333, A 0.000, B 0.000, C 0.000 }
gfCNCPoint1[9681] = {X 132.2366, Y 6.4368, Z -1.3333, A 0.000, B 0.000, C 0.000 }
gfCNCPoint1[9682] = {X 133.1547, Y 6.3238, Z -1.3333, A 0.000, B 0.000, C 0.000 }
gfCNCPoint1[9683] = {X 133.8850, Y 6.3237, Z -1.3333, A 0.000, B 0.000, C 0.000 }
gfCNCPoint1[9684] = {X 134.6956, Y 6.4120, Z -1.3333, A 0.000, B 0.000, C 0.000 }
gfCNCPoint1[9685] = {X 135.4735, Y 6.6567, Z -1.3333, A 0.000, B 0.000, C 0.000 }
gfCNCPoint1[9686] = {X 136.1887, Y 7.0484, Z -1.3333, A 0.000, B 0.000, C 0.000 }
gfCNCPoint1[9687] = {X 136.8137, Y 7.5721, Z -1.3333, A 0.000, B 0.000, C 0.000 }
gfCNCPoint1[9688] = {X 137.3246, Y 8.2077, Z -1.3333, A 0.000, B 0.000, C 0.000 }
gfCNCPoint1[9689] = {X 155.1974, Y 8.2088, Z -1.3333, A 0.000, B 0.000, C 0.000 }
gfCNCPoint1[9690] = {X 155.7090, Y 7.5721, Z -1.3333, A 0.000, B 0.000, C 0.000 }
